 FB 143
BEGIN
   S704_LM_DC_PIN.Enable_Aux := FALSE;
   S704_LM_DC_PIN.Adv_Amount := 0;
   S704_LM_DC_PIN.Ret_Amount := 0;
   S704_LM_DC_PIN.LS_Adv1 := FALSE;
   S704_LM_DC_PIN.LS_Ret1 := FALSE;
   S704_LM_DC_PIN.LS_Adv2 := FALSE;
   S704_LM_DC_PIN.LS_Ret2 := FALSE;
   S704_LM_DC_PIN.LS_Adv3 := FALSE;
   S704_LM_DC_PIN.LS_Ret3 := FALSE;
   S704_LM_DC_PIN.LS_Adv4 := FALSE;
   S704_LM_DC_PIN.LS_Ret4 := FALSE;
   S704_LM_DC_PIN.SOL_Adv := FALSE;
   S704_LM_DC_PIN.SOL_Ret := FALSE;
   S704_LM_DC_PIN.M_Ready := FALSE;
   S704_LM_DC_PIN.T_CHK1 := T#0MS;
   S704_LM_DC_PIN.T_CHK2 := T#0MS;
   S704_LM_DC_PIN.PB_Lamp_CHK := FALSE;
   S704_LM_DC_PIN.PB_Error_Rst := FALSE;
   S704_LM_DC_PIN.M_FLICK := FALSE;
   S704_LM_DC_PIN.M_Adv_Err := FALSE;
   S704_LM_DC_PIN.M_Ret_Err := FALSE;
   S704_LM_DC_PIN.LP_Adv := FALSE;
   S704_LM_DC_PIN.LP_Ret := FALSE;
   S704_LM_DC_PIN.Visu_Adv := W#16#0;
   S704_LM_DC_PIN.Visu_Ret := W#16#0;
   S704_LM_DC_PIN.Error_T1.IN := FALSE;
   S704_LM_DC_PIN.Error_T1.PT := T#0MS;
   S704_LM_DC_PIN.Error_T1.Q := FALSE;
   S704_LM_DC_PIN.Error_T1.ET := T#0MS;
   S704_LM_DC_PIN.Error_T1.STATE := B#16#0;
   S704_LM_DC_PIN.Error_T1.STIME := T#0MS;
   S704_LM_DC_PIN.Error_T1.ATIME := T#0MS;
   S704_LM_DC_PIN.Error_T2.IN := FALSE;
   S704_LM_DC_PIN.Error_T2.PT := T#0MS;
   S704_LM_DC_PIN.Error_T2.Q := FALSE;
   S704_LM_DC_PIN.Error_T2.ET := T#0MS;
   S704_LM_DC_PIN.Error_T2.STATE := B#16#0;
   S704_LM_DC_PIN.Error_T2.STIME := T#0MS;
   S704_LM_DC_PIN.Error_T2.ATIME := T#0MS;
   S704_LM_DC_PIN.CHK_Aux1 := FALSE;
   S704_LM_DC_PIN.CHK_Aux2 := FALSE;
   S704_LM_DC_PIN.Error_T1_DN := FALSE;
   S704_LM_DC_PIN.Error_T2_DN := FALSE;
   S704_LM_DC_PIN.Adv_Memo := FALSE;
   S704_LM_DC_PIN.Visu_Adv_Arr[0] := FALSE;
   S704_LM_DC_PIN.Visu_Adv_Arr[1] := FALSE;
   S704_LM_DC_PIN.Visu_Adv_Arr[2] := FALSE;
   S704_LM_DC_PIN.Visu_Adv_Arr[3] := FALSE;
   S704_LM_DC_PIN.Visu_Adv_Arr[4] := FALSE;
   S704_LM_DC_PIN.Visu_Adv_Arr[5] := FALSE;
   S704_LM_DC_PIN.Visu_Adv_Arr[6] := FALSE;
   S704_LM_DC_PIN.Visu_Adv_Arr[7] := FALSE;
   S704_LM_DC_PIN.Visu_Adv_Arr[8] := FALSE;
   S704_LM_DC_PIN.Visu_Adv_Arr[9] := FALSE;
   S704_LM_DC_PIN.Visu_Adv_Arr[10] := FALSE;
   S704_LM_DC_PIN.Visu_Adv_Arr[11] := FALSE;
   S704_LM_DC_PIN.Visu_Adv_Arr[12] := FALSE;
   S704_LM_DC_PIN.Visu_Adv_Arr[13] := FALSE;
   S704_LM_DC_PIN.Visu_Adv_Arr[14] := FALSE;
   S704_LM_DC_PIN.Visu_Adv_Arr[15] := FALSE;
   S704_LM_DC_PIN.Visu_Ret_Arr[0] := FALSE;
   S704_LM_DC_PIN.Visu_Ret_Arr[1] := FALSE;
   S704_LM_DC_PIN.Visu_Ret_Arr[2] := FALSE;
   S704_LM_DC_PIN.Visu_Ret_Arr[3] := FALSE;
   S704_LM_DC_PIN.Visu_Ret_Arr[4] := FALSE;
   S704_LM_DC_PIN.Visu_Ret_Arr[5] := FALSE;
   S704_LM_DC_PIN.Visu_Ret_Arr[6] := FALSE;
   S704_LM_DC_PIN.Visu_Ret_Arr[7] := FALSE;
   S704_LM_DC_PIN.Visu_Ret_Arr[8] := FALSE;
   S704_LM_DC_PIN.Visu_Ret_Arr[9] := FALSE;
   S704_LM_DC_PIN.Visu_Ret_Arr[10] := FALSE;
   S704_LM_DC_PIN.Visu_Ret_Arr[11] := FALSE;
   S704_LM_DC_PIN.Visu_Ret_Arr[12] := FALSE;
   S704_LM_DC_PIN.Visu_Ret_Arr[13] := FALSE;
   S704_LM_DC_PIN.Visu_Ret_Arr[14] := FALSE;
   S704_LM_DC_PIN.Visu_Ret_Arr[15] := FALSE;
   S704_LM_DC_PIN.BLK_Move_Ret := 0;
   S704_LM_DC_PIN.Enable := FALSE;
   S704_LM_DC_PIN.Adv_End := FALSE;
   S704_LM_DC_PIN.Ret_End := FALSE;
   S704_LM_DC_1ST_CLAMP1.Enable_Aux := FALSE;
   S704_LM_DC_1ST_CLAMP1.Adv_Amount := 0;
   S704_LM_DC_1ST_CLAMP1.Ret_Amount := 0;
   S704_LM_DC_1ST_CLAMP1.LS_Adv1 := FALSE;
   S704_LM_DC_1ST_CLAMP1.LS_Ret1 := FALSE;
   S704_LM_DC_1ST_CLAMP1.LS_Adv2 := FALSE;
   S704_LM_DC_1ST_CLAMP1.LS_Ret2 := FALSE;
   S704_LM_DC_1ST_CLAMP1.LS_Adv3 := FALSE;
   S704_LM_DC_1ST_CLAMP1.LS_Ret3 := FALSE;
   S704_LM_DC_1ST_CLAMP1.LS_Adv4 := FALSE;
   S704_LM_DC_1ST_CLAMP1.LS_Ret4 := FALSE;
   S704_LM_DC_1ST_CLAMP1.SOL_Adv := FALSE;
   S704_LM_DC_1ST_CLAMP1.SOL_Ret := FALSE;
   S704_LM_DC_1ST_CLAMP1.M_Ready := FALSE;
   S704_LM_DC_1ST_CLAMP1.T_CHK1 := T#0MS;
   S704_LM_DC_1ST_CLAMP1.T_CHK2 := T#0MS;
   S704_LM_DC_1ST_CLAMP1.PB_Lamp_CHK := FALSE;
   S704_LM_DC_1ST_CLAMP1.PB_Error_Rst := FALSE;
   S704_LM_DC_1ST_CLAMP1.M_FLICK := FALSE;
   S704_LM_DC_1ST_CLAMP1.M_Adv_Err := FALSE;
   S704_LM_DC_1ST_CLAMP1.M_Ret_Err := FALSE;
   S704_LM_DC_1ST_CLAMP1.LP_Adv := FALSE;
   S704_LM_DC_1ST_CLAMP1.LP_Ret := FALSE;
   S704_LM_DC_1ST_CLAMP1.Visu_Adv := W#16#0;
   S704_LM_DC_1ST_CLAMP1.Visu_Ret := W#16#0;
   S704_LM_DC_1ST_CLAMP1.Error_T1.IN := FALSE;
   S704_LM_DC_1ST_CLAMP1.Error_T1.PT := T#0MS;
   S704_LM_DC_1ST_CLAMP1.Error_T1.Q := FALSE;
   S704_LM_DC_1ST_CLAMP1.Error_T1.ET := T#0MS;
   S704_LM_DC_1ST_CLAMP1.Error_T1.STATE := B#16#0;
   S704_LM_DC_1ST_CLAMP1.Error_T1.STIME := T#0MS;
   S704_LM_DC_1ST_CLAMP1.Error_T1.ATIME := T#0MS;
   S704_LM_DC_1ST_CLAMP1.Error_T2.IN := FALSE;
   S704_LM_DC_1ST_CLAMP1.Error_T2.PT := T#0MS;
   S704_LM_DC_1ST_CLAMP1.Error_T2.Q := FALSE;
   S704_LM_DC_1ST_CLAMP1.Error_T2.ET := T#0MS;
   S704_LM_DC_1ST_CLAMP1.Error_T2.STATE := B#16#0;
   S704_LM_DC_1ST_CLAMP1.Error_T2.STIME := T#0MS;
   S704_LM_DC_1ST_CLAMP1.Error_T2.ATIME := T#0MS;
   S704_LM_DC_1ST_CLAMP1.CHK_Aux1 := FALSE;
   S704_LM_DC_1ST_CLAMP1.CHK_Aux2 := FALSE;
   S704_LM_DC_1ST_CLAMP1.Error_T1_DN := FALSE;
   S704_LM_DC_1ST_CLAMP1.Error_T2_DN := FALSE;
   S704_LM_DC_1ST_CLAMP1.Adv_Memo := FALSE;
   S704_LM_DC_1ST_CLAMP1.Visu_Adv_Arr[0] := FALSE;
   S704_LM_DC_1ST_CLAMP1.Visu_Adv_Arr[1] := FALSE;
   S704_LM_DC_1ST_CLAMP1.Visu_Adv_Arr[2] := FALSE;
   S704_LM_DC_1ST_CLAMP1.Visu_Adv_Arr[3] := FALSE;
   S704_LM_DC_1ST_CLAMP1.Visu_Adv_Arr[4] := FALSE;
   S704_LM_DC_1ST_CLAMP1.Visu_Adv_Arr[5] := FALSE;
   S704_LM_DC_1ST_CLAMP1.Visu_Adv_Arr[6] := FALSE;
   S704_LM_DC_1ST_CLAMP1.Visu_Adv_Arr[7] := FALSE;
   S704_LM_DC_1ST_CLAMP1.Visu_Adv_Arr[8] := FALSE;
   S704_LM_DC_1ST_CLAMP1.Visu_Adv_Arr[9] := FALSE;
   S704_LM_DC_1ST_CLAMP1.Visu_Adv_Arr[10] := FALSE;
   S704_LM_DC_1ST_CLAMP1.Visu_Adv_Arr[11] := FALSE;
   S704_LM_DC_1ST_CLAMP1.Visu_Adv_Arr[12] := FALSE;
   S704_LM_DC_1ST_CLAMP1.Visu_Adv_Arr[13] := FALSE;
   S704_LM_DC_1ST_CLAMP1.Visu_Adv_Arr[14] := FALSE;
   S704_LM_DC_1ST_CLAMP1.Visu_Adv_Arr[15] := FALSE;
   S704_LM_DC_1ST_CLAMP1.Visu_Ret_Arr[0] := FALSE;
   S704_LM_DC_1ST_CLAMP1.Visu_Ret_Arr[1] := FALSE;
   S704_LM_DC_1ST_CLAMP1.Visu_Ret_Arr[2] := FALSE;
   S704_LM_DC_1ST_CLAMP1.Visu_Ret_Arr[3] := FALSE;
   S704_LM_DC_1ST_CLAMP1.Visu_Ret_Arr[4] := FALSE;
   S704_LM_DC_1ST_CLAMP1.Visu_Ret_Arr[5] := FALSE;
   S704_LM_DC_1ST_CLAMP1.Visu_Ret_Arr[6] := FALSE;
   S704_LM_DC_1ST_CLAMP1.Visu_Ret_Arr[7] := FALSE;
   S704_LM_DC_1ST_CLAMP1.Visu_Ret_Arr[8] := FALSE;
   S704_LM_DC_1ST_CLAMP1.Visu_Ret_Arr[9] := FALSE;
   S704_LM_DC_1ST_CLAMP1.Visu_Ret_Arr[10] := FALSE;
   S704_LM_DC_1ST_CLAMP1.Visu_Ret_Arr[11] := FALSE;
   S704_LM_DC_1ST_CLAMP1.Visu_Ret_Arr[12] := FALSE;
   S704_LM_DC_1ST_CLAMP1.Visu_Ret_Arr[13] := FALSE;
   S704_LM_DC_1ST_CLAMP1.Visu_Ret_Arr[14] := FALSE;
   S704_LM_DC_1ST_CLAMP1.Visu_Ret_Arr[15] := FALSE;
   S704_LM_DC_1ST_CLAMP1.BLK_Move_Ret := 0;
   S704_LM_DC_1ST_CLAMP1.Enable := FALSE;
   S704_LM_DC_1ST_CLAMP1.Adv_End := FALSE;
   S704_LM_DC_1ST_CLAMP1.Ret_End := FALSE;
   S704_LM_DC_1ST_CLAMP2.Enable_Aux := FALSE;
   S704_LM_DC_1ST_CLAMP2.Adv_Amount := 0;
   S704_LM_DC_1ST_CLAMP2.Ret_Amount := 0;
   S704_LM_DC_1ST_CLAMP2.LS_Adv1 := FALSE;
   S704_LM_DC_1ST_CLAMP2.LS_Ret1 := FALSE;
   S704_LM_DC_1ST_CLAMP2.LS_Adv2 := FALSE;
   S704_LM_DC_1ST_CLAMP2.LS_Ret2 := FALSE;
   S704_LM_DC_1ST_CLAMP2.LS_Adv3 := FALSE;
   S704_LM_DC_1ST_CLAMP2.LS_Ret3 := FALSE;
   S704_LM_DC_1ST_CLAMP2.LS_Adv4 := FALSE;
   S704_LM_DC_1ST_CLAMP2.LS_Ret4 := FALSE;
   S704_LM_DC_1ST_CLAMP2.SOL_Adv := FALSE;
   S704_LM_DC_1ST_CLAMP2.SOL_Ret := FALSE;
   S704_LM_DC_1ST_CLAMP2.M_Ready := FALSE;
   S704_LM_DC_1ST_CLAMP2.T_CHK1 := T#0MS;
   S704_LM_DC_1ST_CLAMP2.T_CHK2 := T#0MS;
   S704_LM_DC_1ST_CLAMP2.PB_Lamp_CHK := FALSE;
   S704_LM_DC_1ST_CLAMP2.PB_Error_Rst := FALSE;
   S704_LM_DC_1ST_CLAMP2.M_FLICK := FALSE;
   S704_LM_DC_1ST_CLAMP2.M_Adv_Err := FALSE;
   S704_LM_DC_1ST_CLAMP2.M_Ret_Err := FALSE;
   S704_LM_DC_1ST_CLAMP2.LP_Adv := FALSE;
   S704_LM_DC_1ST_CLAMP2.LP_Ret := FALSE;
   S704_LM_DC_1ST_CLAMP2.Visu_Adv := W#16#0;
   S704_LM_DC_1ST_CLAMP2.Visu_Ret := W#16#0;
   S704_LM_DC_1ST_CLAMP2.Error_T1.IN := FALSE;
   S704_LM_DC_1ST_CLAMP2.Error_T1.PT := T#0MS;
   S704_LM_DC_1ST_CLAMP2.Error_T1.Q := FALSE;
   S704_LM_DC_1ST_CLAMP2.Error_T1.ET := T#0MS;
   S704_LM_DC_1ST_CLAMP2.Error_T1.STATE := B#16#0;
   S704_LM_DC_1ST_CLAMP2.Error_T1.STIME := T#0MS;
   S704_LM_DC_1ST_CLAMP2.Error_T1.ATIME := T#0MS;
   S704_LM_DC_1ST_CLAMP2.Error_T2.IN := FALSE;
   S704_LM_DC_1ST_CLAMP2.Error_T2.PT := T#0MS;
   S704_LM_DC_1ST_CLAMP2.Error_T2.Q := FALSE;
   S704_LM_DC_1ST_CLAMP2.Error_T2.ET := T#0MS;
   S704_LM_DC_1ST_CLAMP2.Error_T2.STATE := B#16#0;
   S704_LM_DC_1ST_CLAMP2.Error_T2.STIME := T#0MS;
   S704_LM_DC_1ST_CLAMP2.Error_T2.ATIME := T#0MS;
   S704_LM_DC_1ST_CLAMP2.CHK_Aux1 := FALSE;
   S704_LM_DC_1ST_CLAMP2.CHK_Aux2 := FALSE;
   S704_LM_DC_1ST_CLAMP2.Error_T1_DN := FALSE;
   S704_LM_DC_1ST_CLAMP2.Error_T2_DN := FALSE;
   S704_LM_DC_1ST_CLAMP2.Adv_Memo := FALSE;
   S704_LM_DC_1ST_CLAMP2.Visu_Adv_Arr[0] := FALSE;
   S704_LM_DC_1ST_CLAMP2.Visu_Adv_Arr[1] := FALSE;
   S704_LM_DC_1ST_CLAMP2.Visu_Adv_Arr[2] := FALSE;
   S704_LM_DC_1ST_CLAMP2.Visu_Adv_Arr[3] := FALSE;
   S704_LM_DC_1ST_CLAMP2.Visu_Adv_Arr[4] := FALSE;
   S704_LM_DC_1ST_CLAMP2.Visu_Adv_Arr[5] := FALSE;
   S704_LM_DC_1ST_CLAMP2.Visu_Adv_Arr[6] := FALSE;
   S704_LM_DC_1ST_CLAMP2.Visu_Adv_Arr[7] := FALSE;
   S704_LM_DC_1ST_CLAMP2.Visu_Adv_Arr[8] := FALSE;
   S704_LM_DC_1ST_CLAMP2.Visu_Adv_Arr[9] := FALSE;
   S704_LM_DC_1ST_CLAMP2.Visu_Adv_Arr[10] := FALSE;
   S704_LM_DC_1ST_CLAMP2.Visu_Adv_Arr[11] := FALSE;
   S704_LM_DC_1ST_CLAMP2.Visu_Adv_Arr[12] := FALSE;
   S704_LM_DC_1ST_CLAMP2.Visu_Adv_Arr[13] := FALSE;
   S704_LM_DC_1ST_CLAMP2.Visu_Adv_Arr[14] := FALSE;
   S704_LM_DC_1ST_CLAMP2.Visu_Adv_Arr[15] := FALSE;
   S704_LM_DC_1ST_CLAMP2.Visu_Ret_Arr[0] := FALSE;
   S704_LM_DC_1ST_CLAMP2.Visu_Ret_Arr[1] := FALSE;
   S704_LM_DC_1ST_CLAMP2.Visu_Ret_Arr[2] := FALSE;
   S704_LM_DC_1ST_CLAMP2.Visu_Ret_Arr[3] := FALSE;
   S704_LM_DC_1ST_CLAMP2.Visu_Ret_Arr[4] := FALSE;
   S704_LM_DC_1ST_CLAMP2.Visu_Ret_Arr[5] := FALSE;
   S704_LM_DC_1ST_CLAMP2.Visu_Ret_Arr[6] := FALSE;
   S704_LM_DC_1ST_CLAMP2.Visu_Ret_Arr[7] := FALSE;
   S704_LM_DC_1ST_CLAMP2.Visu_Ret_Arr[8] := FALSE;
   S704_LM_DC_1ST_CLAMP2.Visu_Ret_Arr[9] := FALSE;
   S704_LM_DC_1ST_CLAMP2.Visu_Ret_Arr[10] := FALSE;
   S704_LM_DC_1ST_CLAMP2.Visu_Ret_Arr[11] := FALSE;
   S704_LM_DC_1ST_CLAMP2.Visu_Ret_Arr[12] := FALSE;
   S704_LM_DC_1ST_CLAMP2.Visu_Ret_Arr[13] := FALSE;
   S704_LM_DC_1ST_CLAMP2.Visu_Ret_Arr[14] := FALSE;
   S704_LM_DC_1ST_CLAMP2.Visu_Ret_Arr[15] := FALSE;
   S704_LM_DC_1ST_CLAMP2.BLK_Move_Ret := 0;
   S704_LM_DC_1ST_CLAMP2.Enable := FALSE;
   S704_LM_DC_1ST_CLAMP2.Adv_End := FALSE;
   S704_LM_DC_1ST_CLAMP2.Ret_End := FALSE;
   S704_LM_DC_1ST_CLAMP3.Enable_Aux := FALSE;
   S704_LM_DC_1ST_CLAMP3.Adv_Amount := 0;
   S704_LM_DC_1ST_CLAMP3.Ret_Amount := 0;
   S704_LM_DC_1ST_CLAMP3.LS_Adv1 := FALSE;
   S704_LM_DC_1ST_CLAMP3.LS_Ret1 := FALSE;
   S704_LM_DC_1ST_CLAMP3.LS_Adv2 := FALSE;
   S704_LM_DC_1ST_CLAMP3.LS_Ret2 := FALSE;
   S704_LM_DC_1ST_CLAMP3.LS_Adv3 := FALSE;
   S704_LM_DC_1ST_CLAMP3.LS_Ret3 := FALSE;
   S704_LM_DC_1ST_CLAMP3.LS_Adv4 := FALSE;
   S704_LM_DC_1ST_CLAMP3.LS_Ret4 := FALSE;
   S704_LM_DC_1ST_CLAMP3.SOL_Adv := FALSE;
   S704_LM_DC_1ST_CLAMP3.SOL_Ret := FALSE;
   S704_LM_DC_1ST_CLAMP3.M_Ready := FALSE;
   S704_LM_DC_1ST_CLAMP3.T_CHK1 := T#0MS;
   S704_LM_DC_1ST_CLAMP3.T_CHK2 := T#0MS;
   S704_LM_DC_1ST_CLAMP3.PB_Lamp_CHK := FALSE;
   S704_LM_DC_1ST_CLAMP3.PB_Error_Rst := FALSE;
   S704_LM_DC_1ST_CLAMP3.M_FLICK := FALSE;
   S704_LM_DC_1ST_CLAMP3.M_Adv_Err := FALSE;
   S704_LM_DC_1ST_CLAMP3.M_Ret_Err := FALSE;
   S704_LM_DC_1ST_CLAMP3.LP_Adv := FALSE;
   S704_LM_DC_1ST_CLAMP3.LP_Ret := FALSE;
   S704_LM_DC_1ST_CLAMP3.Visu_Adv := W#16#0;
   S704_LM_DC_1ST_CLAMP3.Visu_Ret := W#16#0;
   S704_LM_DC_1ST_CLAMP3.Error_T1.IN := FALSE;
   S704_LM_DC_1ST_CLAMP3.Error_T1.PT := T#0MS;
   S704_LM_DC_1ST_CLAMP3.Error_T1.Q := FALSE;
   S704_LM_DC_1ST_CLAMP3.Error_T1.ET := T#0MS;
   S704_LM_DC_1ST_CLAMP3.Error_T1.STATE := B#16#0;
   S704_LM_DC_1ST_CLAMP3.Error_T1.STIME := T#0MS;
   S704_LM_DC_1ST_CLAMP3.Error_T1.ATIME := T#0MS;
   S704_LM_DC_1ST_CLAMP3.Error_T2.IN := FALSE;
   S704_LM_DC_1ST_CLAMP3.Error_T2.PT := T#0MS;
   S704_LM_DC_1ST_CLAMP3.Error_T2.Q := FALSE;
   S704_LM_DC_1ST_CLAMP3.Error_T2.ET := T#0MS;
   S704_LM_DC_1ST_CLAMP3.Error_T2.STATE := B#16#0;
   S704_LM_DC_1ST_CLAMP3.Error_T2.STIME := T#0MS;
   S704_LM_DC_1ST_CLAMP3.Error_T2.ATIME := T#0MS;
   S704_LM_DC_1ST_CLAMP3.CHK_Aux1 := FALSE;
   S704_LM_DC_1ST_CLAMP3.CHK_Aux2 := FALSE;
   S704_LM_DC_1ST_CLAMP3.Error_T1_DN := FALSE;
   S704_LM_DC_1ST_CLAMP3.Error_T2_DN := FALSE;
   S704_LM_DC_1ST_CLAMP3.Adv_Memo := FALSE;
   S704_LM_DC_1ST_CLAMP3.Visu_Adv_Arr[0] := FALSE;
   S704_LM_DC_1ST_CLAMP3.Visu_Adv_Arr[1] := FALSE;
   S704_LM_DC_1ST_CLAMP3.Visu_Adv_Arr[2] := FALSE;
   S704_LM_DC_1ST_CLAMP3.Visu_Adv_Arr[3] := FALSE;
   S704_LM_DC_1ST_CLAMP3.Visu_Adv_Arr[4] := FALSE;
   S704_LM_DC_1ST_CLAMP3.Visu_Adv_Arr[5] := FALSE;
   S704_LM_DC_1ST_CLAMP3.Visu_Adv_Arr[6] := FALSE;
   S704_LM_DC_1ST_CLAMP3.Visu_Adv_Arr[7] := FALSE;
   S704_LM_DC_1ST_CLAMP3.Visu_Adv_Arr[8] := FALSE;
   S704_LM_DC_1ST_CLAMP3.Visu_Adv_Arr[9] := FALSE;
   S704_LM_DC_1ST_CLAMP3.Visu_Adv_Arr[10] := FALSE;
   S704_LM_DC_1ST_CLAMP3.Visu_Adv_Arr[11] := FALSE;
   S704_LM_DC_1ST_CLAMP3.Visu_Adv_Arr[12] := FALSE;
   S704_LM_DC_1ST_CLAMP3.Visu_Adv_Arr[13] := FALSE;
   S704_LM_DC_1ST_CLAMP3.Visu_Adv_Arr[14] := FALSE;
   S704_LM_DC_1ST_CLAMP3.Visu_Adv_Arr[15] := FALSE;
   S704_LM_DC_1ST_CLAMP3.Visu_Ret_Arr[0] := FALSE;
   S704_LM_DC_1ST_CLAMP3.Visu_Ret_Arr[1] := FALSE;
   S704_LM_DC_1ST_CLAMP3.Visu_Ret_Arr[2] := FALSE;
   S704_LM_DC_1ST_CLAMP3.Visu_Ret_Arr[3] := FALSE;
   S704_LM_DC_1ST_CLAMP3.Visu_Ret_Arr[4] := FALSE;
   S704_LM_DC_1ST_CLAMP3.Visu_Ret_Arr[5] := FALSE;
   S704_LM_DC_1ST_CLAMP3.Visu_Ret_Arr[6] := FALSE;
   S704_LM_DC_1ST_CLAMP3.Visu_Ret_Arr[7] := FALSE;
   S704_LM_DC_1ST_CLAMP3.Visu_Ret_Arr[8] := FALSE;
   S704_LM_DC_1ST_CLAMP3.Visu_Ret_Arr[9] := FALSE;
   S704_LM_DC_1ST_CLAMP3.Visu_Ret_Arr[10] := FALSE;
   S704_LM_DC_1ST_CLAMP3.Visu_Ret_Arr[11] := FALSE;
   S704_LM_DC_1ST_CLAMP3.Visu_Ret_Arr[12] := FALSE;
   S704_LM_DC_1ST_CLAMP3.Visu_Ret_Arr[13] := FALSE;
   S704_LM_DC_1ST_CLAMP3.Visu_Ret_Arr[14] := FALSE;
   S704_LM_DC_1ST_CLAMP3.Visu_Ret_Arr[15] := FALSE;
   S704_LM_DC_1ST_CLAMP3.BLK_Move_Ret := 0;
   S704_LM_DC_1ST_CLAMP3.Enable := FALSE;
   S704_LM_DC_1ST_CLAMP3.Adv_End := FALSE;
   S704_LM_DC_1ST_CLAMP3.Ret_End := FALSE;
   S704_LM_DC_1ST_CLAMP4.Enable_Aux := FALSE;
   S704_LM_DC_1ST_CLAMP4.Adv_Amount := 0;
   S704_LM_DC_1ST_CLAMP4.Ret_Amount := 0;
   S704_LM_DC_1ST_CLAMP4.LS_Adv1 := FALSE;
   S704_LM_DC_1ST_CLAMP4.LS_Ret1 := FALSE;
   S704_LM_DC_1ST_CLAMP4.LS_Adv2 := FALSE;
   S704_LM_DC_1ST_CLAMP4.LS_Ret2 := FALSE;
   S704_LM_DC_1ST_CLAMP4.LS_Adv3 := FALSE;
   S704_LM_DC_1ST_CLAMP4.LS_Ret3 := FALSE;
   S704_LM_DC_1ST_CLAMP4.LS_Adv4 := FALSE;
   S704_LM_DC_1ST_CLAMP4.LS_Ret4 := FALSE;
   S704_LM_DC_1ST_CLAMP4.SOL_Adv := FALSE;
   S704_LM_DC_1ST_CLAMP4.SOL_Ret := FALSE;
   S704_LM_DC_1ST_CLAMP4.M_Ready := FALSE;
   S704_LM_DC_1ST_CLAMP4.T_CHK1 := T#0MS;
   S704_LM_DC_1ST_CLAMP4.T_CHK2 := T#0MS;
   S704_LM_DC_1ST_CLAMP4.PB_Lamp_CHK := FALSE;
   S704_LM_DC_1ST_CLAMP4.PB_Error_Rst := FALSE;
   S704_LM_DC_1ST_CLAMP4.M_FLICK := FALSE;
   S704_LM_DC_1ST_CLAMP4.M_Adv_Err := FALSE;
   S704_LM_DC_1ST_CLAMP4.M_Ret_Err := FALSE;
   S704_LM_DC_1ST_CLAMP4.LP_Adv := FALSE;
   S704_LM_DC_1ST_CLAMP4.LP_Ret := FALSE;
   S704_LM_DC_1ST_CLAMP4.Visu_Adv := W#16#0;
   S704_LM_DC_1ST_CLAMP4.Visu_Ret := W#16#0;
   S704_LM_DC_1ST_CLAMP4.Error_T1.IN := FALSE;
   S704_LM_DC_1ST_CLAMP4.Error_T1.PT := T#0MS;
   S704_LM_DC_1ST_CLAMP4.Error_T1.Q := FALSE;
   S704_LM_DC_1ST_CLAMP4.Error_T1.ET := T#0MS;
   S704_LM_DC_1ST_CLAMP4.Error_T1.STATE := B#16#0;
   S704_LM_DC_1ST_CLAMP4.Error_T1.STIME := T#0MS;
   S704_LM_DC_1ST_CLAMP4.Error_T1.ATIME := T#0MS;
   S704_LM_DC_1ST_CLAMP4.Error_T2.IN := FALSE;
   S704_LM_DC_1ST_CLAMP4.Error_T2.PT := T#0MS;
   S704_LM_DC_1ST_CLAMP4.Error_T2.Q := FALSE;
   S704_LM_DC_1ST_CLAMP4.Error_T2.ET := T#0MS;
   S704_LM_DC_1ST_CLAMP4.Error_T2.STATE := B#16#0;
   S704_LM_DC_1ST_CLAMP4.Error_T2.STIME := T#0MS;
   S704_LM_DC_1ST_CLAMP4.Error_T2.ATIME := T#0MS;
   S704_LM_DC_1ST_CLAMP4.CHK_Aux1 := FALSE;
   S704_LM_DC_1ST_CLAMP4.CHK_Aux2 := FALSE;
   S704_LM_DC_1ST_CLAMP4.Error_T1_DN := FALSE;
   S704_LM_DC_1ST_CLAMP4.Error_T2_DN := FALSE;
   S704_LM_DC_1ST_CLAMP4.Adv_Memo := FALSE;
   S704_LM_DC_1ST_CLAMP4.Visu_Adv_Arr[0] := FALSE;
   S704_LM_DC_1ST_CLAMP4.Visu_Adv_Arr[1] := FALSE;
   S704_LM_DC_1ST_CLAMP4.Visu_Adv_Arr[2] := FALSE;
   S704_LM_DC_1ST_CLAMP4.Visu_Adv_Arr[3] := FALSE;
   S704_LM_DC_1ST_CLAMP4.Visu_Adv_Arr[4] := FALSE;
   S704_LM_DC_1ST_CLAMP4.Visu_Adv_Arr[5] := FALSE;
   S704_LM_DC_1ST_CLAMP4.Visu_Adv_Arr[6] := FALSE;
   S704_LM_DC_1ST_CLAMP4.Visu_Adv_Arr[7] := FALSE;
   S704_LM_DC_1ST_CLAMP4.Visu_Adv_Arr[8] := FALSE;
   S704_LM_DC_1ST_CLAMP4.Visu_Adv_Arr[9] := FALSE;
   S704_LM_DC_1ST_CLAMP4.Visu_Adv_Arr[10] := FALSE;
   S704_LM_DC_1ST_CLAMP4.Visu_Adv_Arr[11] := FALSE;
   S704_LM_DC_1ST_CLAMP4.Visu_Adv_Arr[12] := FALSE;
   S704_LM_DC_1ST_CLAMP4.Visu_Adv_Arr[13] := FALSE;
   S704_LM_DC_1ST_CLAMP4.Visu_Adv_Arr[14] := FALSE;
   S704_LM_DC_1ST_CLAMP4.Visu_Adv_Arr[15] := FALSE;
   S704_LM_DC_1ST_CLAMP4.Visu_Ret_Arr[0] := FALSE;
   S704_LM_DC_1ST_CLAMP4.Visu_Ret_Arr[1] := FALSE;
   S704_LM_DC_1ST_CLAMP4.Visu_Ret_Arr[2] := FALSE;
   S704_LM_DC_1ST_CLAMP4.Visu_Ret_Arr[3] := FALSE;
   S704_LM_DC_1ST_CLAMP4.Visu_Ret_Arr[4] := FALSE;
   S704_LM_DC_1ST_CLAMP4.Visu_Ret_Arr[5] := FALSE;
   S704_LM_DC_1ST_CLAMP4.Visu_Ret_Arr[6] := FALSE;
   S704_LM_DC_1ST_CLAMP4.Visu_Ret_Arr[7] := FALSE;
   S704_LM_DC_1ST_CLAMP4.Visu_Ret_Arr[8] := FALSE;
   S704_LM_DC_1ST_CLAMP4.Visu_Ret_Arr[9] := FALSE;
   S704_LM_DC_1ST_CLAMP4.Visu_Ret_Arr[10] := FALSE;
   S704_LM_DC_1ST_CLAMP4.Visu_Ret_Arr[11] := FALSE;
   S704_LM_DC_1ST_CLAMP4.Visu_Ret_Arr[12] := FALSE;
   S704_LM_DC_1ST_CLAMP4.Visu_Ret_Arr[13] := FALSE;
   S704_LM_DC_1ST_CLAMP4.Visu_Ret_Arr[14] := FALSE;
   S704_LM_DC_1ST_CLAMP4.Visu_Ret_Arr[15] := FALSE;
   S704_LM_DC_1ST_CLAMP4.BLK_Move_Ret := 0;
   S704_LM_DC_1ST_CLAMP4.Enable := FALSE;
   S704_LM_DC_1ST_CLAMP4.Adv_End := FALSE;
   S704_LM_DC_1ST_CLAMP4.Ret_End := FALSE;
   S704_LM_DC_2ND_CLAMP1.Enable_Aux := FALSE;
   S704_LM_DC_2ND_CLAMP1.Adv_Amount := 0;
   S704_LM_DC_2ND_CLAMP1.Ret_Amount := 0;
   S704_LM_DC_2ND_CLAMP1.LS_Adv1 := FALSE;
   S704_LM_DC_2ND_CLAMP1.LS_Ret1 := FALSE;
   S704_LM_DC_2ND_CLAMP1.LS_Adv2 := FALSE;
   S704_LM_DC_2ND_CLAMP1.LS_Ret2 := FALSE;
   S704_LM_DC_2ND_CLAMP1.LS_Adv3 := FALSE;
   S704_LM_DC_2ND_CLAMP1.LS_Ret3 := FALSE;
   S704_LM_DC_2ND_CLAMP1.LS_Adv4 := FALSE;
   S704_LM_DC_2ND_CLAMP1.LS_Ret4 := FALSE;
   S704_LM_DC_2ND_CLAMP1.SOL_Adv := FALSE;
   S704_LM_DC_2ND_CLAMP1.SOL_Ret := FALSE;
   S704_LM_DC_2ND_CLAMP1.M_Ready := FALSE;
   S704_LM_DC_2ND_CLAMP1.T_CHK1 := T#0MS;
   S704_LM_DC_2ND_CLAMP1.T_CHK2 := T#0MS;
   S704_LM_DC_2ND_CLAMP1.PB_Lamp_CHK := FALSE;
   S704_LM_DC_2ND_CLAMP1.PB_Error_Rst := FALSE;
   S704_LM_DC_2ND_CLAMP1.M_FLICK := FALSE;
   S704_LM_DC_2ND_CLAMP1.M_Adv_Err := FALSE;
   S704_LM_DC_2ND_CLAMP1.M_Ret_Err := FALSE;
   S704_LM_DC_2ND_CLAMP1.LP_Adv := FALSE;
   S704_LM_DC_2ND_CLAMP1.LP_Ret := FALSE;
   S704_LM_DC_2ND_CLAMP1.Visu_Adv := W#16#0;
   S704_LM_DC_2ND_CLAMP1.Visu_Ret := W#16#0;
   S704_LM_DC_2ND_CLAMP1.Error_T1.IN := FALSE;
   S704_LM_DC_2ND_CLAMP1.Error_T1.PT := T#0MS;
   S704_LM_DC_2ND_CLAMP1.Error_T1.Q := FALSE;
   S704_LM_DC_2ND_CLAMP1.Error_T1.ET := T#0MS;
   S704_LM_DC_2ND_CLAMP1.Error_T1.STATE := B#16#0;
   S704_LM_DC_2ND_CLAMP1.Error_T1.STIME := T#0MS;
   S704_LM_DC_2ND_CLAMP1.Error_T1.ATIME := T#0MS;
   S704_LM_DC_2ND_CLAMP1.Error_T2.IN := FALSE;
   S704_LM_DC_2ND_CLAMP1.Error_T2.PT := T#0MS;
   S704_LM_DC_2ND_CLAMP1.Error_T2.Q := FALSE;
   S704_LM_DC_2ND_CLAMP1.Error_T2.ET := T#0MS;
   S704_LM_DC_2ND_CLAMP1.Error_T2.STATE := B#16#0;
   S704_LM_DC_2ND_CLAMP1.Error_T2.STIME := T#0MS;
   S704_LM_DC_2ND_CLAMP1.Error_T2.ATIME := T#0MS;
   S704_LM_DC_2ND_CLAMP1.CHK_Aux1 := FALSE;
   S704_LM_DC_2ND_CLAMP1.CHK_Aux2 := FALSE;
   S704_LM_DC_2ND_CLAMP1.Error_T1_DN := FALSE;
   S704_LM_DC_2ND_CLAMP1.Error_T2_DN := FALSE;
   S704_LM_DC_2ND_CLAMP1.Adv_Memo := FALSE;
   S704_LM_DC_2ND_CLAMP1.Visu_Adv_Arr[0] := FALSE;
   S704_LM_DC_2ND_CLAMP1.Visu_Adv_Arr[1] := FALSE;
   S704_LM_DC_2ND_CLAMP1.Visu_Adv_Arr[2] := FALSE;
   S704_LM_DC_2ND_CLAMP1.Visu_Adv_Arr[3] := FALSE;
   S704_LM_DC_2ND_CLAMP1.Visu_Adv_Arr[4] := FALSE;
   S704_LM_DC_2ND_CLAMP1.Visu_Adv_Arr[5] := FALSE;
   S704_LM_DC_2ND_CLAMP1.Visu_Adv_Arr[6] := FALSE;
   S704_LM_DC_2ND_CLAMP1.Visu_Adv_Arr[7] := FALSE;
   S704_LM_DC_2ND_CLAMP1.Visu_Adv_Arr[8] := FALSE;
   S704_LM_DC_2ND_CLAMP1.Visu_Adv_Arr[9] := FALSE;
   S704_LM_DC_2ND_CLAMP1.Visu_Adv_Arr[10] := FALSE;
   S704_LM_DC_2ND_CLAMP1.Visu_Adv_Arr[11] := FALSE;
   S704_LM_DC_2ND_CLAMP1.Visu_Adv_Arr[12] := FALSE;
   S704_LM_DC_2ND_CLAMP1.Visu_Adv_Arr[13] := FALSE;
   S704_LM_DC_2ND_CLAMP1.Visu_Adv_Arr[14] := FALSE;
   S704_LM_DC_2ND_CLAMP1.Visu_Adv_Arr[15] := FALSE;
   S704_LM_DC_2ND_CLAMP1.Visu_Ret_Arr[0] := FALSE;
   S704_LM_DC_2ND_CLAMP1.Visu_Ret_Arr[1] := FALSE;
   S704_LM_DC_2ND_CLAMP1.Visu_Ret_Arr[2] := FALSE;
   S704_LM_DC_2ND_CLAMP1.Visu_Ret_Arr[3] := FALSE;
   S704_LM_DC_2ND_CLAMP1.Visu_Ret_Arr[4] := FALSE;
   S704_LM_DC_2ND_CLAMP1.Visu_Ret_Arr[5] := FALSE;
   S704_LM_DC_2ND_CLAMP1.Visu_Ret_Arr[6] := FALSE;
   S704_LM_DC_2ND_CLAMP1.Visu_Ret_Arr[7] := FALSE;
   S704_LM_DC_2ND_CLAMP1.Visu_Ret_Arr[8] := FALSE;
   S704_LM_DC_2ND_CLAMP1.Visu_Ret_Arr[9] := FALSE;
   S704_LM_DC_2ND_CLAMP1.Visu_Ret_Arr[10] := FALSE;
   S704_LM_DC_2ND_CLAMP1.Visu_Ret_Arr[11] := FALSE;
   S704_LM_DC_2ND_CLAMP1.Visu_Ret_Arr[12] := FALSE;
   S704_LM_DC_2ND_CLAMP1.Visu_Ret_Arr[13] := FALSE;
   S704_LM_DC_2ND_CLAMP1.Visu_Ret_Arr[14] := FALSE;
   S704_LM_DC_2ND_CLAMP1.Visu_Ret_Arr[15] := FALSE;
   S704_LM_DC_2ND_CLAMP1.BLK_Move_Ret := 0;
   S704_LM_DC_2ND_CLAMP1.Enable := FALSE;
   S704_LM_DC_2ND_CLAMP1.Adv_End := FALSE;
   S704_LM_DC_2ND_CLAMP1.Ret_End := FALSE;
   S704_LM_DC_2ND_CLAMP2.Enable_Aux := FALSE;
   S704_LM_DC_2ND_CLAMP2.Adv_Amount := 0;
   S704_LM_DC_2ND_CLAMP2.Ret_Amount := 0;
   S704_LM_DC_2ND_CLAMP2.LS_Adv1 := FALSE;
   S704_LM_DC_2ND_CLAMP2.LS_Ret1 := FALSE;
   S704_LM_DC_2ND_CLAMP2.LS_Adv2 := FALSE;
   S704_LM_DC_2ND_CLAMP2.LS_Ret2 := FALSE;
   S704_LM_DC_2ND_CLAMP2.LS_Adv3 := FALSE;
   S704_LM_DC_2ND_CLAMP2.LS_Ret3 := FALSE;
   S704_LM_DC_2ND_CLAMP2.LS_Adv4 := FALSE;
   S704_LM_DC_2ND_CLAMP2.LS_Ret4 := FALSE;
   S704_LM_DC_2ND_CLAMP2.SOL_Adv := FALSE;
   S704_LM_DC_2ND_CLAMP2.SOL_Ret := FALSE;
   S704_LM_DC_2ND_CLAMP2.M_Ready := FALSE;
   S704_LM_DC_2ND_CLAMP2.T_CHK1 := T#0MS;
   S704_LM_DC_2ND_CLAMP2.T_CHK2 := T#0MS;
   S704_LM_DC_2ND_CLAMP2.PB_Lamp_CHK := FALSE;
   S704_LM_DC_2ND_CLAMP2.PB_Error_Rst := FALSE;
   S704_LM_DC_2ND_CLAMP2.M_FLICK := FALSE;
   S704_LM_DC_2ND_CLAMP2.M_Adv_Err := FALSE;
   S704_LM_DC_2ND_CLAMP2.M_Ret_Err := FALSE;
   S704_LM_DC_2ND_CLAMP2.LP_Adv := FALSE;
   S704_LM_DC_2ND_CLAMP2.LP_Ret := FALSE;
   S704_LM_DC_2ND_CLAMP2.Visu_Adv := W#16#0;
   S704_LM_DC_2ND_CLAMP2.Visu_Ret := W#16#0;
   S704_LM_DC_2ND_CLAMP2.Error_T1.IN := FALSE;
   S704_LM_DC_2ND_CLAMP2.Error_T1.PT := T#0MS;
   S704_LM_DC_2ND_CLAMP2.Error_T1.Q := FALSE;
   S704_LM_DC_2ND_CLAMP2.Error_T1.ET := T#0MS;
   S704_LM_DC_2ND_CLAMP2.Error_T1.STATE := B#16#0;
   S704_LM_DC_2ND_CLAMP2.Error_T1.STIME := T#0MS;
   S704_LM_DC_2ND_CLAMP2.Error_T1.ATIME := T#0MS;
   S704_LM_DC_2ND_CLAMP2.Error_T2.IN := FALSE;
   S704_LM_DC_2ND_CLAMP2.Error_T2.PT := T#0MS;
   S704_LM_DC_2ND_CLAMP2.Error_T2.Q := FALSE;
   S704_LM_DC_2ND_CLAMP2.Error_T2.ET := T#0MS;
   S704_LM_DC_2ND_CLAMP2.Error_T2.STATE := B#16#0;
   S704_LM_DC_2ND_CLAMP2.Error_T2.STIME := T#0MS;
   S704_LM_DC_2ND_CLAMP2.Error_T2.ATIME := T#0MS;
   S704_LM_DC_2ND_CLAMP2.CHK_Aux1 := FALSE;
   S704_LM_DC_2ND_CLAMP2.CHK_Aux2 := FALSE;
   S704_LM_DC_2ND_CLAMP2.Error_T1_DN := FALSE;
   S704_LM_DC_2ND_CLAMP2.Error_T2_DN := FALSE;
   S704_LM_DC_2ND_CLAMP2.Adv_Memo := FALSE;
   S704_LM_DC_2ND_CLAMP2.Visu_Adv_Arr[0] := FALSE;
   S704_LM_DC_2ND_CLAMP2.Visu_Adv_Arr[1] := FALSE;
   S704_LM_DC_2ND_CLAMP2.Visu_Adv_Arr[2] := FALSE;
   S704_LM_DC_2ND_CLAMP2.Visu_Adv_Arr[3] := FALSE;
   S704_LM_DC_2ND_CLAMP2.Visu_Adv_Arr[4] := FALSE;
   S704_LM_DC_2ND_CLAMP2.Visu_Adv_Arr[5] := FALSE;
   S704_LM_DC_2ND_CLAMP2.Visu_Adv_Arr[6] := FALSE;
   S704_LM_DC_2ND_CLAMP2.Visu_Adv_Arr[7] := FALSE;
   S704_LM_DC_2ND_CLAMP2.Visu_Adv_Arr[8] := FALSE;
   S704_LM_DC_2ND_CLAMP2.Visu_Adv_Arr[9] := FALSE;
   S704_LM_DC_2ND_CLAMP2.Visu_Adv_Arr[10] := FALSE;
   S704_LM_DC_2ND_CLAMP2.Visu_Adv_Arr[11] := FALSE;
   S704_LM_DC_2ND_CLAMP2.Visu_Adv_Arr[12] := FALSE;
   S704_LM_DC_2ND_CLAMP2.Visu_Adv_Arr[13] := FALSE;
   S704_LM_DC_2ND_CLAMP2.Visu_Adv_Arr[14] := FALSE;
   S704_LM_DC_2ND_CLAMP2.Visu_Adv_Arr[15] := FALSE;
   S704_LM_DC_2ND_CLAMP2.Visu_Ret_Arr[0] := FALSE;
   S704_LM_DC_2ND_CLAMP2.Visu_Ret_Arr[1] := FALSE;
   S704_LM_DC_2ND_CLAMP2.Visu_Ret_Arr[2] := FALSE;
   S704_LM_DC_2ND_CLAMP2.Visu_Ret_Arr[3] := FALSE;
   S704_LM_DC_2ND_CLAMP2.Visu_Ret_Arr[4] := FALSE;
   S704_LM_DC_2ND_CLAMP2.Visu_Ret_Arr[5] := FALSE;
   S704_LM_DC_2ND_CLAMP2.Visu_Ret_Arr[6] := FALSE;
   S704_LM_DC_2ND_CLAMP2.Visu_Ret_Arr[7] := FALSE;
   S704_LM_DC_2ND_CLAMP2.Visu_Ret_Arr[8] := FALSE;
   S704_LM_DC_2ND_CLAMP2.Visu_Ret_Arr[9] := FALSE;
   S704_LM_DC_2ND_CLAMP2.Visu_Ret_Arr[10] := FALSE;
   S704_LM_DC_2ND_CLAMP2.Visu_Ret_Arr[11] := FALSE;
   S704_LM_DC_2ND_CLAMP2.Visu_Ret_Arr[12] := FALSE;
   S704_LM_DC_2ND_CLAMP2.Visu_Ret_Arr[13] := FALSE;
   S704_LM_DC_2ND_CLAMP2.Visu_Ret_Arr[14] := FALSE;
   S704_LM_DC_2ND_CLAMP2.Visu_Ret_Arr[15] := FALSE;
   S704_LM_DC_2ND_CLAMP2.BLK_Move_Ret := 0;
   S704_LM_DC_2ND_CLAMP2.Enable := FALSE;
   S704_LM_DC_2ND_CLAMP2.Adv_End := FALSE;
   S704_LM_DC_2ND_CLAMP2.Ret_End := FALSE;
   S704_LM_DC_2ND_CLAMP3.Enable_Aux := FALSE;
   S704_LM_DC_2ND_CLAMP3.Adv_Amount := 0;
   S704_LM_DC_2ND_CLAMP3.Ret_Amount := 0;
   S704_LM_DC_2ND_CLAMP3.LS_Adv1 := FALSE;
   S704_LM_DC_2ND_CLAMP3.LS_Ret1 := FALSE;
   S704_LM_DC_2ND_CLAMP3.LS_Adv2 := FALSE;
   S704_LM_DC_2ND_CLAMP3.LS_Ret2 := FALSE;
   S704_LM_DC_2ND_CLAMP3.LS_Adv3 := FALSE;
   S704_LM_DC_2ND_CLAMP3.LS_Ret3 := FALSE;
   S704_LM_DC_2ND_CLAMP3.LS_Adv4 := FALSE;
   S704_LM_DC_2ND_CLAMP3.LS_Ret4 := FALSE;
   S704_LM_DC_2ND_CLAMP3.SOL_Adv := FALSE;
   S704_LM_DC_2ND_CLAMP3.SOL_Ret := FALSE;
   S704_LM_DC_2ND_CLAMP3.M_Ready := FALSE;
   S704_LM_DC_2ND_CLAMP3.T_CHK1 := T#0MS;
   S704_LM_DC_2ND_CLAMP3.T_CHK2 := T#0MS;
   S704_LM_DC_2ND_CLAMP3.PB_Lamp_CHK := FALSE;
   S704_LM_DC_2ND_CLAMP3.PB_Error_Rst := FALSE;
   S704_LM_DC_2ND_CLAMP3.M_FLICK := FALSE;
   S704_LM_DC_2ND_CLAMP3.M_Adv_Err := FALSE;
   S704_LM_DC_2ND_CLAMP3.M_Ret_Err := FALSE;
   S704_LM_DC_2ND_CLAMP3.LP_Adv := FALSE;
   S704_LM_DC_2ND_CLAMP3.LP_Ret := FALSE;
   S704_LM_DC_2ND_CLAMP3.Visu_Adv := W#16#0;
   S704_LM_DC_2ND_CLAMP3.Visu_Ret := W#16#0;
   S704_LM_DC_2ND_CLAMP3.Error_T1.IN := FALSE;
   S704_LM_DC_2ND_CLAMP3.Error_T1.PT := T#0MS;
   S704_LM_DC_2ND_CLAMP3.Error_T1.Q := FALSE;
   S704_LM_DC_2ND_CLAMP3.Error_T1.ET := T#0MS;
   S704_LM_DC_2ND_CLAMP3.Error_T1.STATE := B#16#0;
   S704_LM_DC_2ND_CLAMP3.Error_T1.STIME := T#0MS;
   S704_LM_DC_2ND_CLAMP3.Error_T1.ATIME := T#0MS;
   S704_LM_DC_2ND_CLAMP3.Error_T2.IN := FALSE;
   S704_LM_DC_2ND_CLAMP3.Error_T2.PT := T#0MS;
   S704_LM_DC_2ND_CLAMP3.Error_T2.Q := FALSE;
   S704_LM_DC_2ND_CLAMP3.Error_T2.ET := T#0MS;
   S704_LM_DC_2ND_CLAMP3.Error_T2.STATE := B#16#0;
   S704_LM_DC_2ND_CLAMP3.Error_T2.STIME := T#0MS;
   S704_LM_DC_2ND_CLAMP3.Error_T2.ATIME := T#0MS;
   S704_LM_DC_2ND_CLAMP3.CHK_Aux1 := FALSE;
   S704_LM_DC_2ND_CLAMP3.CHK_Aux2 := FALSE;
   S704_LM_DC_2ND_CLAMP3.Error_T1_DN := FALSE;
   S704_LM_DC_2ND_CLAMP3.Error_T2_DN := FALSE;
   S704_LM_DC_2ND_CLAMP3.Adv_Memo := FALSE;
   S704_LM_DC_2ND_CLAMP3.Visu_Adv_Arr[0] := FALSE;
   S704_LM_DC_2ND_CLAMP3.Visu_Adv_Arr[1] := FALSE;
   S704_LM_DC_2ND_CLAMP3.Visu_Adv_Arr[2] := FALSE;
   S704_LM_DC_2ND_CLAMP3.Visu_Adv_Arr[3] := FALSE;
   S704_LM_DC_2ND_CLAMP3.Visu_Adv_Arr[4] := FALSE;
   S704_LM_DC_2ND_CLAMP3.Visu_Adv_Arr[5] := FALSE;
   S704_LM_DC_2ND_CLAMP3.Visu_Adv_Arr[6] := FALSE;
   S704_LM_DC_2ND_CLAMP3.Visu_Adv_Arr[7] := FALSE;
   S704_LM_DC_2ND_CLAMP3.Visu_Adv_Arr[8] := FALSE;
   S704_LM_DC_2ND_CLAMP3.Visu_Adv_Arr[9] := FALSE;
   S704_LM_DC_2ND_CLAMP3.Visu_Adv_Arr[10] := FALSE;
   S704_LM_DC_2ND_CLAMP3.Visu_Adv_Arr[11] := FALSE;
   S704_LM_DC_2ND_CLAMP3.Visu_Adv_Arr[12] := FALSE;
   S704_LM_DC_2ND_CLAMP3.Visu_Adv_Arr[13] := FALSE;
   S704_LM_DC_2ND_CLAMP3.Visu_Adv_Arr[14] := FALSE;
   S704_LM_DC_2ND_CLAMP3.Visu_Adv_Arr[15] := FALSE;
   S704_LM_DC_2ND_CLAMP3.Visu_Ret_Arr[0] := FALSE;
   S704_LM_DC_2ND_CLAMP3.Visu_Ret_Arr[1] := FALSE;
   S704_LM_DC_2ND_CLAMP3.Visu_Ret_Arr[2] := FALSE;
   S704_LM_DC_2ND_CLAMP3.Visu_Ret_Arr[3] := FALSE;
   S704_LM_DC_2ND_CLAMP3.Visu_Ret_Arr[4] := FALSE;
   S704_LM_DC_2ND_CLAMP3.Visu_Ret_Arr[5] := FALSE;
   S704_LM_DC_2ND_CLAMP3.Visu_Ret_Arr[6] := FALSE;
   S704_LM_DC_2ND_CLAMP3.Visu_Ret_Arr[7] := FALSE;
   S704_LM_DC_2ND_CLAMP3.Visu_Ret_Arr[8] := FALSE;
   S704_LM_DC_2ND_CLAMP3.Visu_Ret_Arr[9] := FALSE;
   S704_LM_DC_2ND_CLAMP3.Visu_Ret_Arr[10] := FALSE;
   S704_LM_DC_2ND_CLAMP3.Visu_Ret_Arr[11] := FALSE;
   S704_LM_DC_2ND_CLAMP3.Visu_Ret_Arr[12] := FALSE;
   S704_LM_DC_2ND_CLAMP3.Visu_Ret_Arr[13] := FALSE;
   S704_LM_DC_2ND_CLAMP3.Visu_Ret_Arr[14] := FALSE;
   S704_LM_DC_2ND_CLAMP3.Visu_Ret_Arr[15] := FALSE;
   S704_LM_DC_2ND_CLAMP3.BLK_Move_Ret := 0;
   S704_LM_DC_2ND_CLAMP3.Enable := FALSE;
   S704_LM_DC_2ND_CLAMP3.Adv_End := FALSE;
   S704_LM_DC_2ND_CLAMP3.Ret_End := FALSE;
   S704_LM_DC_2ND_CLAMP4.Enable_Aux := FALSE;
   S704_LM_DC_2ND_CLAMP4.Adv_Amount := 0;
   S704_LM_DC_2ND_CLAMP4.Ret_Amount := 0;
   S704_LM_DC_2ND_CLAMP4.LS_Adv1 := FALSE;
   S704_LM_DC_2ND_CLAMP4.LS_Ret1 := FALSE;
   S704_LM_DC_2ND_CLAMP4.LS_Adv2 := FALSE;
   S704_LM_DC_2ND_CLAMP4.LS_Ret2 := FALSE;
   S704_LM_DC_2ND_CLAMP4.LS_Adv3 := FALSE;
   S704_LM_DC_2ND_CLAMP4.LS_Ret3 := FALSE;
   S704_LM_DC_2ND_CLAMP4.LS_Adv4 := FALSE;
   S704_LM_DC_2ND_CLAMP4.LS_Ret4 := FALSE;
   S704_LM_DC_2ND_CLAMP4.SOL_Adv := FALSE;
   S704_LM_DC_2ND_CLAMP4.SOL_Ret := FALSE;
   S704_LM_DC_2ND_CLAMP4.M_Ready := FALSE;
   S704_LM_DC_2ND_CLAMP4.T_CHK1 := T#0MS;
   S704_LM_DC_2ND_CLAMP4.T_CHK2 := T#0MS;
   S704_LM_DC_2ND_CLAMP4.PB_Lamp_CHK := FALSE;
   S704_LM_DC_2ND_CLAMP4.PB_Error_Rst := FALSE;
   S704_LM_DC_2ND_CLAMP4.M_FLICK := FALSE;
   S704_LM_DC_2ND_CLAMP4.M_Adv_Err := FALSE;
   S704_LM_DC_2ND_CLAMP4.M_Ret_Err := FALSE;
   S704_LM_DC_2ND_CLAMP4.LP_Adv := FALSE;
   S704_LM_DC_2ND_CLAMP4.LP_Ret := FALSE;
   S704_LM_DC_2ND_CLAMP4.Visu_Adv := W#16#0;
   S704_LM_DC_2ND_CLAMP4.Visu_Ret := W#16#0;
   S704_LM_DC_2ND_CLAMP4.Error_T1.IN := FALSE;
   S704_LM_DC_2ND_CLAMP4.Error_T1.PT := T#0MS;
   S704_LM_DC_2ND_CLAMP4.Error_T1.Q := FALSE;
   S704_LM_DC_2ND_CLAMP4.Error_T1.ET := T#0MS;
   S704_LM_DC_2ND_CLAMP4.Error_T1.STATE := B#16#0;
   S704_LM_DC_2ND_CLAMP4.Error_T1.STIME := T#0MS;
   S704_LM_DC_2ND_CLAMP4.Error_T1.ATIME := T#0MS;
   S704_LM_DC_2ND_CLAMP4.Error_T2.IN := FALSE;
   S704_LM_DC_2ND_CLAMP4.Error_T2.PT := T#0MS;
   S704_LM_DC_2ND_CLAMP4.Error_T2.Q := FALSE;
   S704_LM_DC_2ND_CLAMP4.Error_T2.ET := T#0MS;
   S704_LM_DC_2ND_CLAMP4.Error_T2.STATE := B#16#0;
   S704_LM_DC_2ND_CLAMP4.Error_T2.STIME := T#0MS;
   S704_LM_DC_2ND_CLAMP4.Error_T2.ATIME := T#0MS;
   S704_LM_DC_2ND_CLAMP4.CHK_Aux1 := FALSE;
   S704_LM_DC_2ND_CLAMP4.CHK_Aux2 := FALSE;
   S704_LM_DC_2ND_CLAMP4.Error_T1_DN := FALSE;
   S704_LM_DC_2ND_CLAMP4.Error_T2_DN := FALSE;
   S704_LM_DC_2ND_CLAMP4.Adv_Memo := FALSE;
   S704_LM_DC_2ND_CLAMP4.Visu_Adv_Arr[0] := FALSE;
   S704_LM_DC_2ND_CLAMP4.Visu_Adv_Arr[1] := FALSE;
   S704_LM_DC_2ND_CLAMP4.Visu_Adv_Arr[2] := FALSE;
   S704_LM_DC_2ND_CLAMP4.Visu_Adv_Arr[3] := FALSE;
   S704_LM_DC_2ND_CLAMP4.Visu_Adv_Arr[4] := FALSE;
   S704_LM_DC_2ND_CLAMP4.Visu_Adv_Arr[5] := FALSE;
   S704_LM_DC_2ND_CLAMP4.Visu_Adv_Arr[6] := FALSE;
   S704_LM_DC_2ND_CLAMP4.Visu_Adv_Arr[7] := FALSE;
   S704_LM_DC_2ND_CLAMP4.Visu_Adv_Arr[8] := FALSE;
   S704_LM_DC_2ND_CLAMP4.Visu_Adv_Arr[9] := FALSE;
   S704_LM_DC_2ND_CLAMP4.Visu_Adv_Arr[10] := FALSE;
   S704_LM_DC_2ND_CLAMP4.Visu_Adv_Arr[11] := FALSE;
   S704_LM_DC_2ND_CLAMP4.Visu_Adv_Arr[12] := FALSE;
   S704_LM_DC_2ND_CLAMP4.Visu_Adv_Arr[13] := FALSE;
   S704_LM_DC_2ND_CLAMP4.Visu_Adv_Arr[14] := FALSE;
   S704_LM_DC_2ND_CLAMP4.Visu_Adv_Arr[15] := FALSE;
   S704_LM_DC_2ND_CLAMP4.Visu_Ret_Arr[0] := FALSE;
   S704_LM_DC_2ND_CLAMP4.Visu_Ret_Arr[1] := FALSE;
   S704_LM_DC_2ND_CLAMP4.Visu_Ret_Arr[2] := FALSE;
   S704_LM_DC_2ND_CLAMP4.Visu_Ret_Arr[3] := FALSE;
   S704_LM_DC_2ND_CLAMP4.Visu_Ret_Arr[4] := FALSE;
   S704_LM_DC_2ND_CLAMP4.Visu_Ret_Arr[5] := FALSE;
   S704_LM_DC_2ND_CLAMP4.Visu_Ret_Arr[6] := FALSE;
   S704_LM_DC_2ND_CLAMP4.Visu_Ret_Arr[7] := FALSE;
   S704_LM_DC_2ND_CLAMP4.Visu_Ret_Arr[8] := FALSE;
   S704_LM_DC_2ND_CLAMP4.Visu_Ret_Arr[9] := FALSE;
   S704_LM_DC_2ND_CLAMP4.Visu_Ret_Arr[10] := FALSE;
   S704_LM_DC_2ND_CLAMP4.Visu_Ret_Arr[11] := FALSE;
   S704_LM_DC_2ND_CLAMP4.Visu_Ret_Arr[12] := FALSE;
   S704_LM_DC_2ND_CLAMP4.Visu_Ret_Arr[13] := FALSE;
   S704_LM_DC_2ND_CLAMP4.Visu_Ret_Arr[14] := FALSE;
   S704_LM_DC_2ND_CLAMP4.Visu_Ret_Arr[15] := FALSE;
   S704_LM_DC_2ND_CLAMP4.BLK_Move_Ret := 0;
   S704_LM_DC_2ND_CLAMP4.Enable := FALSE;
   S704_LM_DC_2ND_CLAMP4.Adv_End := FALSE;
   S704_LM_DC_2ND_CLAMP4.Ret_End := FALSE;
   S704_LM_DC_2ND_CLAMP5.Enable_Aux := FALSE;
   S704_LM_DC_2ND_CLAMP5.Adv_Amount := 0;
   S704_LM_DC_2ND_CLAMP5.Ret_Amount := 0;
   S704_LM_DC_2ND_CLAMP5.LS_Adv1 := FALSE;
   S704_LM_DC_2ND_CLAMP5.LS_Ret1 := FALSE;
   S704_LM_DC_2ND_CLAMP5.LS_Adv2 := FALSE;
   S704_LM_DC_2ND_CLAMP5.LS_Ret2 := FALSE;
   S704_LM_DC_2ND_CLAMP5.LS_Adv3 := FALSE;
   S704_LM_DC_2ND_CLAMP5.LS_Ret3 := FALSE;
   S704_LM_DC_2ND_CLAMP5.LS_Adv4 := FALSE;
   S704_LM_DC_2ND_CLAMP5.LS_Ret4 := FALSE;
   S704_LM_DC_2ND_CLAMP5.SOL_Adv := FALSE;
   S704_LM_DC_2ND_CLAMP5.SOL_Ret := FALSE;
   S704_LM_DC_2ND_CLAMP5.M_Ready := FALSE;
   S704_LM_DC_2ND_CLAMP5.T_CHK1 := T#0MS;
   S704_LM_DC_2ND_CLAMP5.T_CHK2 := T#0MS;
   S704_LM_DC_2ND_CLAMP5.PB_Lamp_CHK := FALSE;
   S704_LM_DC_2ND_CLAMP5.PB_Error_Rst := FALSE;
   S704_LM_DC_2ND_CLAMP5.M_FLICK := FALSE;
   S704_LM_DC_2ND_CLAMP5.M_Adv_Err := FALSE;
   S704_LM_DC_2ND_CLAMP5.M_Ret_Err := FALSE;
   S704_LM_DC_2ND_CLAMP5.LP_Adv := FALSE;
   S704_LM_DC_2ND_CLAMP5.LP_Ret := FALSE;
   S704_LM_DC_2ND_CLAMP5.Visu_Adv := W#16#0;
   S704_LM_DC_2ND_CLAMP5.Visu_Ret := W#16#0;
   S704_LM_DC_2ND_CLAMP5.Error_T1.IN := FALSE;
   S704_LM_DC_2ND_CLAMP5.Error_T1.PT := T#0MS;
   S704_LM_DC_2ND_CLAMP5.Error_T1.Q := FALSE;
   S704_LM_DC_2ND_CLAMP5.Error_T1.ET := T#0MS;
   S704_LM_DC_2ND_CLAMP5.Error_T1.STATE := B#16#0;
   S704_LM_DC_2ND_CLAMP5.Error_T1.STIME := T#0MS;
   S704_LM_DC_2ND_CLAMP5.Error_T1.ATIME := T#0MS;
   S704_LM_DC_2ND_CLAMP5.Error_T2.IN := FALSE;
   S704_LM_DC_2ND_CLAMP5.Error_T2.PT := T#0MS;
   S704_LM_DC_2ND_CLAMP5.Error_T2.Q := FALSE;
   S704_LM_DC_2ND_CLAMP5.Error_T2.ET := T#0MS;
   S704_LM_DC_2ND_CLAMP5.Error_T2.STATE := B#16#0;
   S704_LM_DC_2ND_CLAMP5.Error_T2.STIME := T#0MS;
   S704_LM_DC_2ND_CLAMP5.Error_T2.ATIME := T#0MS;
   S704_LM_DC_2ND_CLAMP5.CHK_Aux1 := FALSE;
   S704_LM_DC_2ND_CLAMP5.CHK_Aux2 := FALSE;
   S704_LM_DC_2ND_CLAMP5.Error_T1_DN := FALSE;
   S704_LM_DC_2ND_CLAMP5.Error_T2_DN := FALSE;
   S704_LM_DC_2ND_CLAMP5.Adv_Memo := FALSE;
   S704_LM_DC_2ND_CLAMP5.Visu_Adv_Arr[0] := FALSE;
   S704_LM_DC_2ND_CLAMP5.Visu_Adv_Arr[1] := FALSE;
   S704_LM_DC_2ND_CLAMP5.Visu_Adv_Arr[2] := FALSE;
   S704_LM_DC_2ND_CLAMP5.Visu_Adv_Arr[3] := FALSE;
   S704_LM_DC_2ND_CLAMP5.Visu_Adv_Arr[4] := FALSE;
   S704_LM_DC_2ND_CLAMP5.Visu_Adv_Arr[5] := FALSE;
   S704_LM_DC_2ND_CLAMP5.Visu_Adv_Arr[6] := FALSE;
   S704_LM_DC_2ND_CLAMP5.Visu_Adv_Arr[7] := FALSE;
   S704_LM_DC_2ND_CLAMP5.Visu_Adv_Arr[8] := FALSE;
   S704_LM_DC_2ND_CLAMP5.Visu_Adv_Arr[9] := FALSE;
   S704_LM_DC_2ND_CLAMP5.Visu_Adv_Arr[10] := FALSE;
   S704_LM_DC_2ND_CLAMP5.Visu_Adv_Arr[11] := FALSE;
   S704_LM_DC_2ND_CLAMP5.Visu_Adv_Arr[12] := FALSE;
   S704_LM_DC_2ND_CLAMP5.Visu_Adv_Arr[13] := FALSE;
   S704_LM_DC_2ND_CLAMP5.Visu_Adv_Arr[14] := FALSE;
   S704_LM_DC_2ND_CLAMP5.Visu_Adv_Arr[15] := FALSE;
   S704_LM_DC_2ND_CLAMP5.Visu_Ret_Arr[0] := FALSE;
   S704_LM_DC_2ND_CLAMP5.Visu_Ret_Arr[1] := FALSE;
   S704_LM_DC_2ND_CLAMP5.Visu_Ret_Arr[2] := FALSE;
   S704_LM_DC_2ND_CLAMP5.Visu_Ret_Arr[3] := FALSE;
   S704_LM_DC_2ND_CLAMP5.Visu_Ret_Arr[4] := FALSE;
   S704_LM_DC_2ND_CLAMP5.Visu_Ret_Arr[5] := FALSE;
   S704_LM_DC_2ND_CLAMP5.Visu_Ret_Arr[6] := FALSE;
   S704_LM_DC_2ND_CLAMP5.Visu_Ret_Arr[7] := FALSE;
   S704_LM_DC_2ND_CLAMP5.Visu_Ret_Arr[8] := FALSE;
   S704_LM_DC_2ND_CLAMP5.Visu_Ret_Arr[9] := FALSE;
   S704_LM_DC_2ND_CLAMP5.Visu_Ret_Arr[10] := FALSE;
   S704_LM_DC_2ND_CLAMP5.Visu_Ret_Arr[11] := FALSE;
   S704_LM_DC_2ND_CLAMP5.Visu_Ret_Arr[12] := FALSE;
   S704_LM_DC_2ND_CLAMP5.Visu_Ret_Arr[13] := FALSE;
   S704_LM_DC_2ND_CLAMP5.Visu_Ret_Arr[14] := FALSE;
   S704_LM_DC_2ND_CLAMP5.Visu_Ret_Arr[15] := FALSE;
   S704_LM_DC_2ND_CLAMP5.BLK_Move_Ret := 0;
   S704_LM_DC_2ND_CLAMP5.Enable := FALSE;
   S704_LM_DC_2ND_CLAMP5.Adv_End := FALSE;
   S704_LM_DC_2ND_CLAMP5.Ret_End := FALSE;
   S704_LM_DC_STK_PIN.Enable_Aux := FALSE;
   S704_LM_DC_STK_PIN.Adv_Amount := 0;
   S704_LM_DC_STK_PIN.Ret_Amount := 0;
   S704_LM_DC_STK_PIN.LS_Adv1 := FALSE;
   S704_LM_DC_STK_PIN.LS_Ret1 := FALSE;
   S704_LM_DC_STK_PIN.LS_Adv2 := FALSE;
   S704_LM_DC_STK_PIN.LS_Ret2 := FALSE;
   S704_LM_DC_STK_PIN.LS_Adv3 := FALSE;
   S704_LM_DC_STK_PIN.LS_Ret3 := FALSE;
   S704_LM_DC_STK_PIN.LS_Adv4 := FALSE;
   S704_LM_DC_STK_PIN.LS_Ret4 := FALSE;
   S704_LM_DC_STK_PIN.SOL_Adv := FALSE;
   S704_LM_DC_STK_PIN.SOL_Ret := FALSE;
   S704_LM_DC_STK_PIN.M_Ready := FALSE;
   S704_LM_DC_STK_PIN.T_CHK1 := T#0MS;
   S704_LM_DC_STK_PIN.T_CHK2 := T#0MS;
   S704_LM_DC_STK_PIN.PB_Lamp_CHK := FALSE;
   S704_LM_DC_STK_PIN.PB_Error_Rst := FALSE;
   S704_LM_DC_STK_PIN.M_FLICK := FALSE;
   S704_LM_DC_STK_PIN.M_Adv_Err := FALSE;
   S704_LM_DC_STK_PIN.M_Ret_Err := FALSE;
   S704_LM_DC_STK_PIN.LP_Adv := FALSE;
   S704_LM_DC_STK_PIN.LP_Ret := FALSE;
   S704_LM_DC_STK_PIN.Visu_Adv := W#16#0;
   S704_LM_DC_STK_PIN.Visu_Ret := W#16#0;
   S704_LM_DC_STK_PIN.Error_T1.IN := FALSE;
   S704_LM_DC_STK_PIN.Error_T1.PT := T#0MS;
   S704_LM_DC_STK_PIN.Error_T1.Q := FALSE;
   S704_LM_DC_STK_PIN.Error_T1.ET := T#0MS;
   S704_LM_DC_STK_PIN.Error_T1.STATE := B#16#0;
   S704_LM_DC_STK_PIN.Error_T1.STIME := T#0MS;
   S704_LM_DC_STK_PIN.Error_T1.ATIME := T#0MS;
   S704_LM_DC_STK_PIN.Error_T2.IN := FALSE;
   S704_LM_DC_STK_PIN.Error_T2.PT := T#0MS;
   S704_LM_DC_STK_PIN.Error_T2.Q := FALSE;
   S704_LM_DC_STK_PIN.Error_T2.ET := T#0MS;
   S704_LM_DC_STK_PIN.Error_T2.STATE := B#16#0;
   S704_LM_DC_STK_PIN.Error_T2.STIME := T#0MS;
   S704_LM_DC_STK_PIN.Error_T2.ATIME := T#0MS;
   S704_LM_DC_STK_PIN.CHK_Aux1 := FALSE;
   S704_LM_DC_STK_PIN.CHK_Aux2 := FALSE;
   S704_LM_DC_STK_PIN.Error_T1_DN := FALSE;
   S704_LM_DC_STK_PIN.Error_T2_DN := FALSE;
   S704_LM_DC_STK_PIN.Adv_Memo := FALSE;
   S704_LM_DC_STK_PIN.Visu_Adv_Arr[0] := FALSE;
   S704_LM_DC_STK_PIN.Visu_Adv_Arr[1] := FALSE;
   S704_LM_DC_STK_PIN.Visu_Adv_Arr[2] := FALSE;
   S704_LM_DC_STK_PIN.Visu_Adv_Arr[3] := FALSE;
   S704_LM_DC_STK_PIN.Visu_Adv_Arr[4] := FALSE;
   S704_LM_DC_STK_PIN.Visu_Adv_Arr[5] := FALSE;
   S704_LM_DC_STK_PIN.Visu_Adv_Arr[6] := FALSE;
   S704_LM_DC_STK_PIN.Visu_Adv_Arr[7] := FALSE;
   S704_LM_DC_STK_PIN.Visu_Adv_Arr[8] := FALSE;
   S704_LM_DC_STK_PIN.Visu_Adv_Arr[9] := FALSE;
   S704_LM_DC_STK_PIN.Visu_Adv_Arr[10] := FALSE;
   S704_LM_DC_STK_PIN.Visu_Adv_Arr[11] := FALSE;
   S704_LM_DC_STK_PIN.Visu_Adv_Arr[12] := FALSE;
   S704_LM_DC_STK_PIN.Visu_Adv_Arr[13] := FALSE;
   S704_LM_DC_STK_PIN.Visu_Adv_Arr[14] := FALSE;
   S704_LM_DC_STK_PIN.Visu_Adv_Arr[15] := FALSE;
   S704_LM_DC_STK_PIN.Visu_Ret_Arr[0] := FALSE;
   S704_LM_DC_STK_PIN.Visu_Ret_Arr[1] := FALSE;
   S704_LM_DC_STK_PIN.Visu_Ret_Arr[2] := FALSE;
   S704_LM_DC_STK_PIN.Visu_Ret_Arr[3] := FALSE;
   S704_LM_DC_STK_PIN.Visu_Ret_Arr[4] := FALSE;
   S704_LM_DC_STK_PIN.Visu_Ret_Arr[5] := FALSE;
   S704_LM_DC_STK_PIN.Visu_Ret_Arr[6] := FALSE;
   S704_LM_DC_STK_PIN.Visu_Ret_Arr[7] := FALSE;
   S704_LM_DC_STK_PIN.Visu_Ret_Arr[8] := FALSE;
   S704_LM_DC_STK_PIN.Visu_Ret_Arr[9] := FALSE;
   S704_LM_DC_STK_PIN.Visu_Ret_Arr[10] := FALSE;
   S704_LM_DC_STK_PIN.Visu_Ret_Arr[11] := FALSE;
   S704_LM_DC_STK_PIN.Visu_Ret_Arr[12] := FALSE;
   S704_LM_DC_STK_PIN.Visu_Ret_Arr[13] := FALSE;
   S704_LM_DC_STK_PIN.Visu_Ret_Arr[14] := FALSE;
   S704_LM_DC_STK_PIN.Visu_Ret_Arr[15] := FALSE;
   S704_LM_DC_STK_PIN.BLK_Move_Ret := 0;
   S704_LM_DC_STK_PIN.Enable := FALSE;
   S704_LM_DC_STK_PIN.Adv_End := FALSE;
   S704_LM_DC_STK_PIN.Ret_End := FALSE;
   S704_LM_DC_OTR_CLAMP.Enable_Aux := FALSE;
   S704_LM_DC_OTR_CLAMP.Adv_Amount := 0;
   S704_LM_DC_OTR_CLAMP.Ret_Amount := 0;
   S704_LM_DC_OTR_CLAMP.LS_Adv1 := FALSE;
   S704_LM_DC_OTR_CLAMP.LS_Ret1 := FALSE;
   S704_LM_DC_OTR_CLAMP.LS_Adv2 := FALSE;
   S704_LM_DC_OTR_CLAMP.LS_Ret2 := FALSE;
   S704_LM_DC_OTR_CLAMP.LS_Adv3 := FALSE;
   S704_LM_DC_OTR_CLAMP.LS_Ret3 := FALSE;
   S704_LM_DC_OTR_CLAMP.LS_Adv4 := FALSE;
   S704_LM_DC_OTR_CLAMP.LS_Ret4 := FALSE;
   S704_LM_DC_OTR_CLAMP.SOL_Adv := FALSE;
   S704_LM_DC_OTR_CLAMP.SOL_Ret := FALSE;
   S704_LM_DC_OTR_CLAMP.M_Ready := FALSE;
   S704_LM_DC_OTR_CLAMP.T_CHK1 := T#0MS;
   S704_LM_DC_OTR_CLAMP.T_CHK2 := T#0MS;
   S704_LM_DC_OTR_CLAMP.PB_Lamp_CHK := FALSE;
   S704_LM_DC_OTR_CLAMP.PB_Error_Rst := FALSE;
   S704_LM_DC_OTR_CLAMP.M_FLICK := FALSE;
   S704_LM_DC_OTR_CLAMP.M_Adv_Err := FALSE;
   S704_LM_DC_OTR_CLAMP.M_Ret_Err := FALSE;
   S704_LM_DC_OTR_CLAMP.LP_Adv := FALSE;
   S704_LM_DC_OTR_CLAMP.LP_Ret := FALSE;
   S704_LM_DC_OTR_CLAMP.Visu_Adv := W#16#0;
   S704_LM_DC_OTR_CLAMP.Visu_Ret := W#16#0;
   S704_LM_DC_OTR_CLAMP.Error_T1.IN := FALSE;
   S704_LM_DC_OTR_CLAMP.Error_T1.PT := T#0MS;
   S704_LM_DC_OTR_CLAMP.Error_T1.Q := FALSE;
   S704_LM_DC_OTR_CLAMP.Error_T1.ET := T#0MS;
   S704_LM_DC_OTR_CLAMP.Error_T1.STATE := B#16#0;
   S704_LM_DC_OTR_CLAMP.Error_T1.STIME := T#0MS;
   S704_LM_DC_OTR_CLAMP.Error_T1.ATIME := T#0MS;
   S704_LM_DC_OTR_CLAMP.Error_T2.IN := FALSE;
   S704_LM_DC_OTR_CLAMP.Error_T2.PT := T#0MS;
   S704_LM_DC_OTR_CLAMP.Error_T2.Q := FALSE;
   S704_LM_DC_OTR_CLAMP.Error_T2.ET := T#0MS;
   S704_LM_DC_OTR_CLAMP.Error_T2.STATE := B#16#0;
   S704_LM_DC_OTR_CLAMP.Error_T2.STIME := T#0MS;
   S704_LM_DC_OTR_CLAMP.Error_T2.ATIME := T#0MS;
   S704_LM_DC_OTR_CLAMP.CHK_Aux1 := FALSE;
   S704_LM_DC_OTR_CLAMP.CHK_Aux2 := FALSE;
   S704_LM_DC_OTR_CLAMP.Error_T1_DN := FALSE;
   S704_LM_DC_OTR_CLAMP.Error_T2_DN := FALSE;
   S704_LM_DC_OTR_CLAMP.Adv_Memo := FALSE;
   S704_LM_DC_OTR_CLAMP.Visu_Adv_Arr[0] := FALSE;
   S704_LM_DC_OTR_CLAMP.Visu_Adv_Arr[1] := FALSE;
   S704_LM_DC_OTR_CLAMP.Visu_Adv_Arr[2] := FALSE;
   S704_LM_DC_OTR_CLAMP.Visu_Adv_Arr[3] := FALSE;
   S704_LM_DC_OTR_CLAMP.Visu_Adv_Arr[4] := FALSE;
   S704_LM_DC_OTR_CLAMP.Visu_Adv_Arr[5] := FALSE;
   S704_LM_DC_OTR_CLAMP.Visu_Adv_Arr[6] := FALSE;
   S704_LM_DC_OTR_CLAMP.Visu_Adv_Arr[7] := FALSE;
   S704_LM_DC_OTR_CLAMP.Visu_Adv_Arr[8] := FALSE;
   S704_LM_DC_OTR_CLAMP.Visu_Adv_Arr[9] := FALSE;
   S704_LM_DC_OTR_CLAMP.Visu_Adv_Arr[10] := FALSE;
   S704_LM_DC_OTR_CLAMP.Visu_Adv_Arr[11] := FALSE;
   S704_LM_DC_OTR_CLAMP.Visu_Adv_Arr[12] := FALSE;
   S704_LM_DC_OTR_CLAMP.Visu_Adv_Arr[13] := FALSE;
   S704_LM_DC_OTR_CLAMP.Visu_Adv_Arr[14] := FALSE;
   S704_LM_DC_OTR_CLAMP.Visu_Adv_Arr[15] := FALSE;
   S704_LM_DC_OTR_CLAMP.Visu_Ret_Arr[0] := FALSE;
   S704_LM_DC_OTR_CLAMP.Visu_Ret_Arr[1] := FALSE;
   S704_LM_DC_OTR_CLAMP.Visu_Ret_Arr[2] := FALSE;
   S704_LM_DC_OTR_CLAMP.Visu_Ret_Arr[3] := FALSE;
   S704_LM_DC_OTR_CLAMP.Visu_Ret_Arr[4] := FALSE;
   S704_LM_DC_OTR_CLAMP.Visu_Ret_Arr[5] := FALSE;
   S704_LM_DC_OTR_CLAMP.Visu_Ret_Arr[6] := FALSE;
   S704_LM_DC_OTR_CLAMP.Visu_Ret_Arr[7] := FALSE;
   S704_LM_DC_OTR_CLAMP.Visu_Ret_Arr[8] := FALSE;
   S704_LM_DC_OTR_CLAMP.Visu_Ret_Arr[9] := FALSE;
   S704_LM_DC_OTR_CLAMP.Visu_Ret_Arr[10] := FALSE;
   S704_LM_DC_OTR_CLAMP.Visu_Ret_Arr[11] := FALSE;
   S704_LM_DC_OTR_CLAMP.Visu_Ret_Arr[12] := FALSE;
   S704_LM_DC_OTR_CLAMP.Visu_Ret_Arr[13] := FALSE;
   S704_LM_DC_OTR_CLAMP.Visu_Ret_Arr[14] := FALSE;
   S704_LM_DC_OTR_CLAMP.Visu_Ret_Arr[15] := FALSE;
   S704_LM_DC_OTR_CLAMP.BLK_Move_Ret := 0;
   S704_LM_DC_OTR_CLAMP.Enable := FALSE;
   S704_LM_DC_OTR_CLAMP.Adv_End := FALSE;
   S704_LM_DC_OTR_CLAMP.Ret_End := FALSE;
   S704_LM_DC_ASSY_CLAMP.Enable_Aux := FALSE;
   S704_LM_DC_ASSY_CLAMP.Adv_Amount := 0;
   S704_LM_DC_ASSY_CLAMP.Ret_Amount := 0;
   S704_LM_DC_ASSY_CLAMP.LS_Adv1 := FALSE;
   S704_LM_DC_ASSY_CLAMP.LS_Ret1 := FALSE;
   S704_LM_DC_ASSY_CLAMP.LS_Adv2 := FALSE;
   S704_LM_DC_ASSY_CLAMP.LS_Ret2 := FALSE;
   S704_LM_DC_ASSY_CLAMP.LS_Adv3 := FALSE;
   S704_LM_DC_ASSY_CLAMP.LS_Ret3 := FALSE;
   S704_LM_DC_ASSY_CLAMP.LS_Adv4 := FALSE;
   S704_LM_DC_ASSY_CLAMP.LS_Ret4 := FALSE;
   S704_LM_DC_ASSY_CLAMP.SOL_Adv := FALSE;
   S704_LM_DC_ASSY_CLAMP.SOL_Ret := FALSE;
   S704_LM_DC_ASSY_CLAMP.M_Ready := FALSE;
   S704_LM_DC_ASSY_CLAMP.T_CHK1 := T#0MS;
   S704_LM_DC_ASSY_CLAMP.T_CHK2 := T#0MS;
   S704_LM_DC_ASSY_CLAMP.PB_Lamp_CHK := FALSE;
   S704_LM_DC_ASSY_CLAMP.PB_Error_Rst := FALSE;
   S704_LM_DC_ASSY_CLAMP.M_FLICK := FALSE;
   S704_LM_DC_ASSY_CLAMP.M_Adv_Err := FALSE;
   S704_LM_DC_ASSY_CLAMP.M_Ret_Err := FALSE;
   S704_LM_DC_ASSY_CLAMP.LP_Adv := FALSE;
   S704_LM_DC_ASSY_CLAMP.LP_Ret := FALSE;
   S704_LM_DC_ASSY_CLAMP.Visu_Adv := W#16#0;
   S704_LM_DC_ASSY_CLAMP.Visu_Ret := W#16#0;
   S704_LM_DC_ASSY_CLAMP.Error_T1.IN := FALSE;
   S704_LM_DC_ASSY_CLAMP.Error_T1.PT := T#0MS;
   S704_LM_DC_ASSY_CLAMP.Error_T1.Q := FALSE;
   S704_LM_DC_ASSY_CLAMP.Error_T1.ET := T#0MS;
   S704_LM_DC_ASSY_CLAMP.Error_T1.STATE := B#16#0;
   S704_LM_DC_ASSY_CLAMP.Error_T1.STIME := T#0MS;
   S704_LM_DC_ASSY_CLAMP.Error_T1.ATIME := T#0MS;
   S704_LM_DC_ASSY_CLAMP.Error_T2.IN := FALSE;
   S704_LM_DC_ASSY_CLAMP.Error_T2.PT := T#0MS;
   S704_LM_DC_ASSY_CLAMP.Error_T2.Q := FALSE;
   S704_LM_DC_ASSY_CLAMP.Error_T2.ET := T#0MS;
   S704_LM_DC_ASSY_CLAMP.Error_T2.STATE := B#16#0;
   S704_LM_DC_ASSY_CLAMP.Error_T2.STIME := T#0MS;
   S704_LM_DC_ASSY_CLAMP.Error_T2.ATIME := T#0MS;
   S704_LM_DC_ASSY_CLAMP.CHK_Aux1 := FALSE;
   S704_LM_DC_ASSY_CLAMP.CHK_Aux2 := FALSE;
   S704_LM_DC_ASSY_CLAMP.Error_T1_DN := FALSE;
   S704_LM_DC_ASSY_CLAMP.Error_T2_DN := FALSE;
   S704_LM_DC_ASSY_CLAMP.Adv_Memo := FALSE;
   S704_LM_DC_ASSY_CLAMP.Visu_Adv_Arr[0] := FALSE;
   S704_LM_DC_ASSY_CLAMP.Visu_Adv_Arr[1] := FALSE;
   S704_LM_DC_ASSY_CLAMP.Visu_Adv_Arr[2] := FALSE;
   S704_LM_DC_ASSY_CLAMP.Visu_Adv_Arr[3] := FALSE;
   S704_LM_DC_ASSY_CLAMP.Visu_Adv_Arr[4] := FALSE;
   S704_LM_DC_ASSY_CLAMP.Visu_Adv_Arr[5] := FALSE;
   S704_LM_DC_ASSY_CLAMP.Visu_Adv_Arr[6] := FALSE;
   S704_LM_DC_ASSY_CLAMP.Visu_Adv_Arr[7] := FALSE;
   S704_LM_DC_ASSY_CLAMP.Visu_Adv_Arr[8] := FALSE;
   S704_LM_DC_ASSY_CLAMP.Visu_Adv_Arr[9] := FALSE;
   S704_LM_DC_ASSY_CLAMP.Visu_Adv_Arr[10] := FALSE;
   S704_LM_DC_ASSY_CLAMP.Visu_Adv_Arr[11] := FALSE;
   S704_LM_DC_ASSY_CLAMP.Visu_Adv_Arr[12] := FALSE;
   S704_LM_DC_ASSY_CLAMP.Visu_Adv_Arr[13] := FALSE;
   S704_LM_DC_ASSY_CLAMP.Visu_Adv_Arr[14] := FALSE;
   S704_LM_DC_ASSY_CLAMP.Visu_Adv_Arr[15] := FALSE;
   S704_LM_DC_ASSY_CLAMP.Visu_Ret_Arr[0] := FALSE;
   S704_LM_DC_ASSY_CLAMP.Visu_Ret_Arr[1] := FALSE;
   S704_LM_DC_ASSY_CLAMP.Visu_Ret_Arr[2] := FALSE;
   S704_LM_DC_ASSY_CLAMP.Visu_Ret_Arr[3] := FALSE;
   S704_LM_DC_ASSY_CLAMP.Visu_Ret_Arr[4] := FALSE;
   S704_LM_DC_ASSY_CLAMP.Visu_Ret_Arr[5] := FALSE;
   S704_LM_DC_ASSY_CLAMP.Visu_Ret_Arr[6] := FALSE;
   S704_LM_DC_ASSY_CLAMP.Visu_Ret_Arr[7] := FALSE;
   S704_LM_DC_ASSY_CLAMP.Visu_Ret_Arr[8] := FALSE;
   S704_LM_DC_ASSY_CLAMP.Visu_Ret_Arr[9] := FALSE;
   S704_LM_DC_ASSY_CLAMP.Visu_Ret_Arr[10] := FALSE;
   S704_LM_DC_ASSY_CLAMP.Visu_Ret_Arr[11] := FALSE;
   S704_LM_DC_ASSY_CLAMP.Visu_Ret_Arr[12] := FALSE;
   S704_LM_DC_ASSY_CLAMP.Visu_Ret_Arr[13] := FALSE;
   S704_LM_DC_ASSY_CLAMP.Visu_Ret_Arr[14] := FALSE;
   S704_LM_DC_ASSY_CLAMP.Visu_Ret_Arr[15] := FALSE;
   S704_LM_DC_ASSY_CLAMP.BLK_Move_Ret := 0;
   S704_LM_DC_ASSY_CLAMP.Enable := FALSE;
   S704_LM_DC_ASSY_CLAMP.Adv_End := FALSE;
   S704_LM_DC_ASSY_CLAMP.Ret_End := FALSE;
   S704_LM_DC_FF_PIN.Enable_Aux := FALSE;
   S704_LM_DC_FF_PIN.Adv_Amount := 0;
   S704_LM_DC_FF_PIN.Ret_Amount := 0;
   S704_LM_DC_FF_PIN.LS_Adv1 := FALSE;
   S704_LM_DC_FF_PIN.LS_Ret1 := FALSE;
   S704_LM_DC_FF_PIN.LS_Adv2 := FALSE;
   S704_LM_DC_FF_PIN.LS_Ret2 := FALSE;
   S704_LM_DC_FF_PIN.LS_Adv3 := FALSE;
   S704_LM_DC_FF_PIN.LS_Ret3 := FALSE;
   S704_LM_DC_FF_PIN.LS_Adv4 := FALSE;
   S704_LM_DC_FF_PIN.LS_Ret4 := FALSE;
   S704_LM_DC_FF_PIN.SOL_Adv := FALSE;
   S704_LM_DC_FF_PIN.SOL_Ret := FALSE;
   S704_LM_DC_FF_PIN.M_Ready := FALSE;
   S704_LM_DC_FF_PIN.T_CHK1 := T#0MS;
   S704_LM_DC_FF_PIN.T_CHK2 := T#0MS;
   S704_LM_DC_FF_PIN.PB_Lamp_CHK := FALSE;
   S704_LM_DC_FF_PIN.PB_Error_Rst := FALSE;
   S704_LM_DC_FF_PIN.M_FLICK := FALSE;
   S704_LM_DC_FF_PIN.M_Adv_Err := FALSE;
   S704_LM_DC_FF_PIN.M_Ret_Err := FALSE;
   S704_LM_DC_FF_PIN.LP_Adv := FALSE;
   S704_LM_DC_FF_PIN.LP_Ret := FALSE;
   S704_LM_DC_FF_PIN.Visu_Adv := W#16#0;
   S704_LM_DC_FF_PIN.Visu_Ret := W#16#0;
   S704_LM_DC_FF_PIN.Error_T1.IN := FALSE;
   S704_LM_DC_FF_PIN.Error_T1.PT := T#0MS;
   S704_LM_DC_FF_PIN.Error_T1.Q := FALSE;
   S704_LM_DC_FF_PIN.Error_T1.ET := T#0MS;
   S704_LM_DC_FF_PIN.Error_T1.STATE := B#16#0;
   S704_LM_DC_FF_PIN.Error_T1.STIME := T#0MS;
   S704_LM_DC_FF_PIN.Error_T1.ATIME := T#0MS;
   S704_LM_DC_FF_PIN.Error_T2.IN := FALSE;
   S704_LM_DC_FF_PIN.Error_T2.PT := T#0MS;
   S704_LM_DC_FF_PIN.Error_T2.Q := FALSE;
   S704_LM_DC_FF_PIN.Error_T2.ET := T#0MS;
   S704_LM_DC_FF_PIN.Error_T2.STATE := B#16#0;
   S704_LM_DC_FF_PIN.Error_T2.STIME := T#0MS;
   S704_LM_DC_FF_PIN.Error_T2.ATIME := T#0MS;
   S704_LM_DC_FF_PIN.CHK_Aux1 := FALSE;
   S704_LM_DC_FF_PIN.CHK_Aux2 := FALSE;
   S704_LM_DC_FF_PIN.Error_T1_DN := FALSE;
   S704_LM_DC_FF_PIN.Error_T2_DN := FALSE;
   S704_LM_DC_FF_PIN.Adv_Memo := FALSE;
   S704_LM_DC_FF_PIN.Visu_Adv_Arr[0] := FALSE;
   S704_LM_DC_FF_PIN.Visu_Adv_Arr[1] := FALSE;
   S704_LM_DC_FF_PIN.Visu_Adv_Arr[2] := FALSE;
   S704_LM_DC_FF_PIN.Visu_Adv_Arr[3] := FALSE;
   S704_LM_DC_FF_PIN.Visu_Adv_Arr[4] := FALSE;
   S704_LM_DC_FF_PIN.Visu_Adv_Arr[5] := FALSE;
   S704_LM_DC_FF_PIN.Visu_Adv_Arr[6] := FALSE;
   S704_LM_DC_FF_PIN.Visu_Adv_Arr[7] := FALSE;
   S704_LM_DC_FF_PIN.Visu_Adv_Arr[8] := FALSE;
   S704_LM_DC_FF_PIN.Visu_Adv_Arr[9] := FALSE;
   S704_LM_DC_FF_PIN.Visu_Adv_Arr[10] := FALSE;
   S704_LM_DC_FF_PIN.Visu_Adv_Arr[11] := FALSE;
   S704_LM_DC_FF_PIN.Visu_Adv_Arr[12] := FALSE;
   S704_LM_DC_FF_PIN.Visu_Adv_Arr[13] := FALSE;
   S704_LM_DC_FF_PIN.Visu_Adv_Arr[14] := FALSE;
   S704_LM_DC_FF_PIN.Visu_Adv_Arr[15] := FALSE;
   S704_LM_DC_FF_PIN.Visu_Ret_Arr[0] := FALSE;
   S704_LM_DC_FF_PIN.Visu_Ret_Arr[1] := FALSE;
   S704_LM_DC_FF_PIN.Visu_Ret_Arr[2] := FALSE;
   S704_LM_DC_FF_PIN.Visu_Ret_Arr[3] := FALSE;
   S704_LM_DC_FF_PIN.Visu_Ret_Arr[4] := FALSE;
   S704_LM_DC_FF_PIN.Visu_Ret_Arr[5] := FALSE;
   S704_LM_DC_FF_PIN.Visu_Ret_Arr[6] := FALSE;
   S704_LM_DC_FF_PIN.Visu_Ret_Arr[7] := FALSE;
   S704_LM_DC_FF_PIN.Visu_Ret_Arr[8] := FALSE;
   S704_LM_DC_FF_PIN.Visu_Ret_Arr[9] := FALSE;
   S704_LM_DC_FF_PIN.Visu_Ret_Arr[10] := FALSE;
   S704_LM_DC_FF_PIN.Visu_Ret_Arr[11] := FALSE;
   S704_LM_DC_FF_PIN.Visu_Ret_Arr[12] := FALSE;
   S704_LM_DC_FF_PIN.Visu_Ret_Arr[13] := FALSE;
   S704_LM_DC_FF_PIN.Visu_Ret_Arr[14] := FALSE;
   S704_LM_DC_FF_PIN.Visu_Ret_Arr[15] := FALSE;
   S704_LM_DC_FF_PIN.BLK_Move_Ret := 0;
   S704_LM_DC_FF_PIN.Enable := FALSE;
   S704_LM_DC_FF_PIN.Adv_End := FALSE;
   S704_LM_DC_FF_PIN.Ret_End := FALSE;
   S704_LM_DC_FF_CLAMP.Enable_Aux := FALSE;
   S704_LM_DC_FF_CLAMP.Adv_Amount := 0;
   S704_LM_DC_FF_CLAMP.Ret_Amount := 0;
   S704_LM_DC_FF_CLAMP.LS_Adv1 := FALSE;
   S704_LM_DC_FF_CLAMP.LS_Ret1 := FALSE;
   S704_LM_DC_FF_CLAMP.LS_Adv2 := FALSE;
   S704_LM_DC_FF_CLAMP.LS_Ret2 := FALSE;
   S704_LM_DC_FF_CLAMP.LS_Adv3 := FALSE;
   S704_LM_DC_FF_CLAMP.LS_Ret3 := FALSE;
   S704_LM_DC_FF_CLAMP.LS_Adv4 := FALSE;
   S704_LM_DC_FF_CLAMP.LS_Ret4 := FALSE;
   S704_LM_DC_FF_CLAMP.SOL_Adv := FALSE;
   S704_LM_DC_FF_CLAMP.SOL_Ret := FALSE;
   S704_LM_DC_FF_CLAMP.M_Ready := FALSE;
   S704_LM_DC_FF_CLAMP.T_CHK1 := T#0MS;
   S704_LM_DC_FF_CLAMP.T_CHK2 := T#0MS;
   S704_LM_DC_FF_CLAMP.PB_Lamp_CHK := FALSE;
   S704_LM_DC_FF_CLAMP.PB_Error_Rst := FALSE;
   S704_LM_DC_FF_CLAMP.M_FLICK := FALSE;
   S704_LM_DC_FF_CLAMP.M_Adv_Err := FALSE;
   S704_LM_DC_FF_CLAMP.M_Ret_Err := FALSE;
   S704_LM_DC_FF_CLAMP.LP_Adv := FALSE;
   S704_LM_DC_FF_CLAMP.LP_Ret := FALSE;
   S704_LM_DC_FF_CLAMP.Visu_Adv := W#16#0;
   S704_LM_DC_FF_CLAMP.Visu_Ret := W#16#0;
   S704_LM_DC_FF_CLAMP.Error_T1.IN := FALSE;
   S704_LM_DC_FF_CLAMP.Error_T1.PT := T#0MS;
   S704_LM_DC_FF_CLAMP.Error_T1.Q := FALSE;
   S704_LM_DC_FF_CLAMP.Error_T1.ET := T#0MS;
   S704_LM_DC_FF_CLAMP.Error_T1.STATE := B#16#0;
   S704_LM_DC_FF_CLAMP.Error_T1.STIME := T#0MS;
   S704_LM_DC_FF_CLAMP.Error_T1.ATIME := T#0MS;
   S704_LM_DC_FF_CLAMP.Error_T2.IN := FALSE;
   S704_LM_DC_FF_CLAMP.Error_T2.PT := T#0MS;
   S704_LM_DC_FF_CLAMP.Error_T2.Q := FALSE;
   S704_LM_DC_FF_CLAMP.Error_T2.ET := T#0MS;
   S704_LM_DC_FF_CLAMP.Error_T2.STATE := B#16#0;
   S704_LM_DC_FF_CLAMP.Error_T2.STIME := T#0MS;
   S704_LM_DC_FF_CLAMP.Error_T2.ATIME := T#0MS;
   S704_LM_DC_FF_CLAMP.CHK_Aux1 := FALSE;
   S704_LM_DC_FF_CLAMP.CHK_Aux2 := FALSE;
   S704_LM_DC_FF_CLAMP.Error_T1_DN := FALSE;
   S704_LM_DC_FF_CLAMP.Error_T2_DN := FALSE;
   S704_LM_DC_FF_CLAMP.Adv_Memo := FALSE;
   S704_LM_DC_FF_CLAMP.Visu_Adv_Arr[0] := FALSE;
   S704_LM_DC_FF_CLAMP.Visu_Adv_Arr[1] := FALSE;
   S704_LM_DC_FF_CLAMP.Visu_Adv_Arr[2] := FALSE;
   S704_LM_DC_FF_CLAMP.Visu_Adv_Arr[3] := FALSE;
   S704_LM_DC_FF_CLAMP.Visu_Adv_Arr[4] := FALSE;
   S704_LM_DC_FF_CLAMP.Visu_Adv_Arr[5] := FALSE;
   S704_LM_DC_FF_CLAMP.Visu_Adv_Arr[6] := FALSE;
   S704_LM_DC_FF_CLAMP.Visu_Adv_Arr[7] := FALSE;
   S704_LM_DC_FF_CLAMP.Visu_Adv_Arr[8] := FALSE;
   S704_LM_DC_FF_CLAMP.Visu_Adv_Arr[9] := FALSE;
   S704_LM_DC_FF_CLAMP.Visu_Adv_Arr[10] := FALSE;
   S704_LM_DC_FF_CLAMP.Visu_Adv_Arr[11] := FALSE;
   S704_LM_DC_FF_CLAMP.Visu_Adv_Arr[12] := FALSE;
   S704_LM_DC_FF_CLAMP.Visu_Adv_Arr[13] := FALSE;
   S704_LM_DC_FF_CLAMP.Visu_Adv_Arr[14] := FALSE;
   S704_LM_DC_FF_CLAMP.Visu_Adv_Arr[15] := FALSE;
   S704_LM_DC_FF_CLAMP.Visu_Ret_Arr[0] := FALSE;
   S704_LM_DC_FF_CLAMP.Visu_Ret_Arr[1] := FALSE;
   S704_LM_DC_FF_CLAMP.Visu_Ret_Arr[2] := FALSE;
   S704_LM_DC_FF_CLAMP.Visu_Ret_Arr[3] := FALSE;
   S704_LM_DC_FF_CLAMP.Visu_Ret_Arr[4] := FALSE;
   S704_LM_DC_FF_CLAMP.Visu_Ret_Arr[5] := FALSE;
   S704_LM_DC_FF_CLAMP.Visu_Ret_Arr[6] := FALSE;
   S704_LM_DC_FF_CLAMP.Visu_Ret_Arr[7] := FALSE;
   S704_LM_DC_FF_CLAMP.Visu_Ret_Arr[8] := FALSE;
   S704_LM_DC_FF_CLAMP.Visu_Ret_Arr[9] := FALSE;
   S704_LM_DC_FF_CLAMP.Visu_Ret_Arr[10] := FALSE;
   S704_LM_DC_FF_CLAMP.Visu_Ret_Arr[11] := FALSE;
   S704_LM_DC_FF_CLAMP.Visu_Ret_Arr[12] := FALSE;
   S704_LM_DC_FF_CLAMP.Visu_Ret_Arr[13] := FALSE;
   S704_LM_DC_FF_CLAMP.Visu_Ret_Arr[14] := FALSE;
   S704_LM_DC_FF_CLAMP.Visu_Ret_Arr[15] := FALSE;
   S704_LM_DC_FF_CLAMP.BLK_Move_Ret := 0;
   S704_LM_DC_FF_CLAMP.Enable := FALSE;
   S704_LM_DC_FF_CLAMP.Adv_End := FALSE;
   S704_LM_DC_FF_CLAMP.Ret_End := FALSE;
   S704_LM_DC_2ND_CLAMP6.Enable_Aux := FALSE;
   S704_LM_DC_2ND_CLAMP6.Adv_Amount := 0;
   S704_LM_DC_2ND_CLAMP6.Ret_Amount := 0;
   S704_LM_DC_2ND_CLAMP6.LS_Adv1 := FALSE;
   S704_LM_DC_2ND_CLAMP6.LS_Ret1 := FALSE;
   S704_LM_DC_2ND_CLAMP6.LS_Adv2 := FALSE;
   S704_LM_DC_2ND_CLAMP6.LS_Ret2 := FALSE;
   S704_LM_DC_2ND_CLAMP6.LS_Adv3 := FALSE;
   S704_LM_DC_2ND_CLAMP6.LS_Ret3 := FALSE;
   S704_LM_DC_2ND_CLAMP6.LS_Adv4 := FALSE;
   S704_LM_DC_2ND_CLAMP6.LS_Ret4 := FALSE;
   S704_LM_DC_2ND_CLAMP6.SOL_Adv := FALSE;
   S704_LM_DC_2ND_CLAMP6.SOL_Ret := FALSE;
   S704_LM_DC_2ND_CLAMP6.M_Ready := FALSE;
   S704_LM_DC_2ND_CLAMP6.T_CHK1 := T#0MS;
   S704_LM_DC_2ND_CLAMP6.T_CHK2 := T#0MS;
   S704_LM_DC_2ND_CLAMP6.PB_Lamp_CHK := FALSE;
   S704_LM_DC_2ND_CLAMP6.PB_Error_Rst := FALSE;
   S704_LM_DC_2ND_CLAMP6.M_FLICK := FALSE;
   S704_LM_DC_2ND_CLAMP6.M_Adv_Err := FALSE;
   S704_LM_DC_2ND_CLAMP6.M_Ret_Err := FALSE;
   S704_LM_DC_2ND_CLAMP6.LP_Adv := FALSE;
   S704_LM_DC_2ND_CLAMP6.LP_Ret := FALSE;
   S704_LM_DC_2ND_CLAMP6.Visu_Adv := W#16#0;
   S704_LM_DC_2ND_CLAMP6.Visu_Ret := W#16#0;
   S704_LM_DC_2ND_CLAMP6.Error_T1.IN := FALSE;
   S704_LM_DC_2ND_CLAMP6.Error_T1.PT := T#0MS;
   S704_LM_DC_2ND_CLAMP6.Error_T1.Q := FALSE;
   S704_LM_DC_2ND_CLAMP6.Error_T1.ET := T#0MS;
   S704_LM_DC_2ND_CLAMP6.Error_T1.STATE := B#16#0;
   S704_LM_DC_2ND_CLAMP6.Error_T1.STIME := T#0MS;
   S704_LM_DC_2ND_CLAMP6.Error_T1.ATIME := T#0MS;
   S704_LM_DC_2ND_CLAMP6.Error_T2.IN := FALSE;
   S704_LM_DC_2ND_CLAMP6.Error_T2.PT := T#0MS;
   S704_LM_DC_2ND_CLAMP6.Error_T2.Q := FALSE;
   S704_LM_DC_2ND_CLAMP6.Error_T2.ET := T#0MS;
   S704_LM_DC_2ND_CLAMP6.Error_T2.STATE := B#16#0;
   S704_LM_DC_2ND_CLAMP6.Error_T2.STIME := T#0MS;
   S704_LM_DC_2ND_CLAMP6.Error_T2.ATIME := T#0MS;
   S704_LM_DC_2ND_CLAMP6.CHK_Aux1 := FALSE;
   S704_LM_DC_2ND_CLAMP6.CHK_Aux2 := FALSE;
   S704_LM_DC_2ND_CLAMP6.Error_T1_DN := FALSE;
   S704_LM_DC_2ND_CLAMP6.Error_T2_DN := FALSE;
   S704_LM_DC_2ND_CLAMP6.Adv_Memo := FALSE;
   S704_LM_DC_2ND_CLAMP6.Visu_Adv_Arr[0] := FALSE;
   S704_LM_DC_2ND_CLAMP6.Visu_Adv_Arr[1] := FALSE;
   S704_LM_DC_2ND_CLAMP6.Visu_Adv_Arr[2] := FALSE;
   S704_LM_DC_2ND_CLAMP6.Visu_Adv_Arr[3] := FALSE;
   S704_LM_DC_2ND_CLAMP6.Visu_Adv_Arr[4] := FALSE;
   S704_LM_DC_2ND_CLAMP6.Visu_Adv_Arr[5] := FALSE;
   S704_LM_DC_2ND_CLAMP6.Visu_Adv_Arr[6] := FALSE;
   S704_LM_DC_2ND_CLAMP6.Visu_Adv_Arr[7] := FALSE;
   S704_LM_DC_2ND_CLAMP6.Visu_Adv_Arr[8] := FALSE;
   S704_LM_DC_2ND_CLAMP6.Visu_Adv_Arr[9] := FALSE;
   S704_LM_DC_2ND_CLAMP6.Visu_Adv_Arr[10] := FALSE;
   S704_LM_DC_2ND_CLAMP6.Visu_Adv_Arr[11] := FALSE;
   S704_LM_DC_2ND_CLAMP6.Visu_Adv_Arr[12] := FALSE;
   S704_LM_DC_2ND_CLAMP6.Visu_Adv_Arr[13] := FALSE;
   S704_LM_DC_2ND_CLAMP6.Visu_Adv_Arr[14] := FALSE;
   S704_LM_DC_2ND_CLAMP6.Visu_Adv_Arr[15] := FALSE;
   S704_LM_DC_2ND_CLAMP6.Visu_Ret_Arr[0] := FALSE;
   S704_LM_DC_2ND_CLAMP6.Visu_Ret_Arr[1] := FALSE;
   S704_LM_DC_2ND_CLAMP6.Visu_Ret_Arr[2] := FALSE;
   S704_LM_DC_2ND_CLAMP6.Visu_Ret_Arr[3] := FALSE;
   S704_LM_DC_2ND_CLAMP6.Visu_Ret_Arr[4] := FALSE;
   S704_LM_DC_2ND_CLAMP6.Visu_Ret_Arr[5] := FALSE;
   S704_LM_DC_2ND_CLAMP6.Visu_Ret_Arr[6] := FALSE;
   S704_LM_DC_2ND_CLAMP6.Visu_Ret_Arr[7] := FALSE;
   S704_LM_DC_2ND_CLAMP6.Visu_Ret_Arr[8] := FALSE;
   S704_LM_DC_2ND_CLAMP6.Visu_Ret_Arr[9] := FALSE;
   S704_LM_DC_2ND_CLAMP6.Visu_Ret_Arr[10] := FALSE;
   S704_LM_DC_2ND_CLAMP6.Visu_Ret_Arr[11] := FALSE;
   S704_LM_DC_2ND_CLAMP6.Visu_Ret_Arr[12] := FALSE;
   S704_LM_DC_2ND_CLAMP6.Visu_Ret_Arr[13] := FALSE;
   S704_LM_DC_2ND_CLAMP6.Visu_Ret_Arr[14] := FALSE;
   S704_LM_DC_2ND_CLAMP6.Visu_Ret_Arr[15] := FALSE;
   S704_LM_DC_2ND_CLAMP6.BLK_Move_Ret := 0;
   S704_LM_DC_2ND_CLAMP6.Enable := FALSE;
   S704_LM_DC_2ND_CLAMP6.Adv_End := FALSE;
   S704_LM_DC_2ND_CLAMP6.Ret_End := FALSE;
   S704_LM_DC_2ND_CLAMP7.Enable_Aux := FALSE;
   S704_LM_DC_2ND_CLAMP7.Adv_Amount := 0;
   S704_LM_DC_2ND_CLAMP7.Ret_Amount := 0;
   S704_LM_DC_2ND_CLAMP7.LS_Adv1 := FALSE;
   S704_LM_DC_2ND_CLAMP7.LS_Ret1 := FALSE;
   S704_LM_DC_2ND_CLAMP7.LS_Adv2 := FALSE;
   S704_LM_DC_2ND_CLAMP7.LS_Ret2 := FALSE;
   S704_LM_DC_2ND_CLAMP7.LS_Adv3 := FALSE;
   S704_LM_DC_2ND_CLAMP7.LS_Ret3 := FALSE;
   S704_LM_DC_2ND_CLAMP7.LS_Adv4 := FALSE;
   S704_LM_DC_2ND_CLAMP7.LS_Ret4 := FALSE;
   S704_LM_DC_2ND_CLAMP7.SOL_Adv := FALSE;
   S704_LM_DC_2ND_CLAMP7.SOL_Ret := FALSE;
   S704_LM_DC_2ND_CLAMP7.M_Ready := FALSE;
   S704_LM_DC_2ND_CLAMP7.T_CHK1 := T#0MS;
   S704_LM_DC_2ND_CLAMP7.T_CHK2 := T#0MS;
   S704_LM_DC_2ND_CLAMP7.PB_Lamp_CHK := FALSE;
   S704_LM_DC_2ND_CLAMP7.PB_Error_Rst := FALSE;
   S704_LM_DC_2ND_CLAMP7.M_FLICK := FALSE;
   S704_LM_DC_2ND_CLAMP7.M_Adv_Err := FALSE;
   S704_LM_DC_2ND_CLAMP7.M_Ret_Err := FALSE;
   S704_LM_DC_2ND_CLAMP7.LP_Adv := FALSE;
   S704_LM_DC_2ND_CLAMP7.LP_Ret := FALSE;
   S704_LM_DC_2ND_CLAMP7.Visu_Adv := W#16#0;
   S704_LM_DC_2ND_CLAMP7.Visu_Ret := W#16#0;
   S704_LM_DC_2ND_CLAMP7.Error_T1.IN := FALSE;
   S704_LM_DC_2ND_CLAMP7.Error_T1.PT := T#0MS;
   S704_LM_DC_2ND_CLAMP7.Error_T1.Q := FALSE;
   S704_LM_DC_2ND_CLAMP7.Error_T1.ET := T#0MS;
   S704_LM_DC_2ND_CLAMP7.Error_T1.STATE := B#16#0;
   S704_LM_DC_2ND_CLAMP7.Error_T1.STIME := T#0MS;
   S704_LM_DC_2ND_CLAMP7.Error_T1.ATIME := T#0MS;
   S704_LM_DC_2ND_CLAMP7.Error_T2.IN := FALSE;
   S704_LM_DC_2ND_CLAMP7.Error_T2.PT := T#0MS;
   S704_LM_DC_2ND_CLAMP7.Error_T2.Q := FALSE;
   S704_LM_DC_2ND_CLAMP7.Error_T2.ET := T#0MS;
   S704_LM_DC_2ND_CLAMP7.Error_T2.STATE := B#16#0;
   S704_LM_DC_2ND_CLAMP7.Error_T2.STIME := T#0MS;
   S704_LM_DC_2ND_CLAMP7.Error_T2.ATIME := T#0MS;
   S704_LM_DC_2ND_CLAMP7.CHK_Aux1 := FALSE;
   S704_LM_DC_2ND_CLAMP7.CHK_Aux2 := FALSE;
   S704_LM_DC_2ND_CLAMP7.Error_T1_DN := FALSE;
   S704_LM_DC_2ND_CLAMP7.Error_T2_DN := FALSE;
   S704_LM_DC_2ND_CLAMP7.Adv_Memo := FALSE;
   S704_LM_DC_2ND_CLAMP7.Visu_Adv_Arr[0] := FALSE;
   S704_LM_DC_2ND_CLAMP7.Visu_Adv_Arr[1] := FALSE;
   S704_LM_DC_2ND_CLAMP7.Visu_Adv_Arr[2] := FALSE;
   S704_LM_DC_2ND_CLAMP7.Visu_Adv_Arr[3] := FALSE;
   S704_LM_DC_2ND_CLAMP7.Visu_Adv_Arr[4] := FALSE;
   S704_LM_DC_2ND_CLAMP7.Visu_Adv_Arr[5] := FALSE;
   S704_LM_DC_2ND_CLAMP7.Visu_Adv_Arr[6] := FALSE;
   S704_LM_DC_2ND_CLAMP7.Visu_Adv_Arr[7] := FALSE;
   S704_LM_DC_2ND_CLAMP7.Visu_Adv_Arr[8] := FALSE;
   S704_LM_DC_2ND_CLAMP7.Visu_Adv_Arr[9] := FALSE;
   S704_LM_DC_2ND_CLAMP7.Visu_Adv_Arr[10] := FALSE;
   S704_LM_DC_2ND_CLAMP7.Visu_Adv_Arr[11] := FALSE;
   S704_LM_DC_2ND_CLAMP7.Visu_Adv_Arr[12] := FALSE;
   S704_LM_DC_2ND_CLAMP7.Visu_Adv_Arr[13] := FALSE;
   S704_LM_DC_2ND_CLAMP7.Visu_Adv_Arr[14] := FALSE;
   S704_LM_DC_2ND_CLAMP7.Visu_Adv_Arr[15] := FALSE;
   S704_LM_DC_2ND_CLAMP7.Visu_Ret_Arr[0] := FALSE;
   S704_LM_DC_2ND_CLAMP7.Visu_Ret_Arr[1] := FALSE;
   S704_LM_DC_2ND_CLAMP7.Visu_Ret_Arr[2] := FALSE;
   S704_LM_DC_2ND_CLAMP7.Visu_Ret_Arr[3] := FALSE;
   S704_LM_DC_2ND_CLAMP7.Visu_Ret_Arr[4] := FALSE;
   S704_LM_DC_2ND_CLAMP7.Visu_Ret_Arr[5] := FALSE;
   S704_LM_DC_2ND_CLAMP7.Visu_Ret_Arr[6] := FALSE;
   S704_LM_DC_2ND_CLAMP7.Visu_Ret_Arr[7] := FALSE;
   S704_LM_DC_2ND_CLAMP7.Visu_Ret_Arr[8] := FALSE;
   S704_LM_DC_2ND_CLAMP7.Visu_Ret_Arr[9] := FALSE;
   S704_LM_DC_2ND_CLAMP7.Visu_Ret_Arr[10] := FALSE;
   S704_LM_DC_2ND_CLAMP7.Visu_Ret_Arr[11] := FALSE;
   S704_LM_DC_2ND_CLAMP7.Visu_Ret_Arr[12] := FALSE;
   S704_LM_DC_2ND_CLAMP7.Visu_Ret_Arr[13] := FALSE;
   S704_LM_DC_2ND_CLAMP7.Visu_Ret_Arr[14] := FALSE;
   S704_LM_DC_2ND_CLAMP7.Visu_Ret_Arr[15] := FALSE;
   S704_LM_DC_2ND_CLAMP7.BLK_Move_Ret := 0;
   S704_LM_DC_2ND_CLAMP7.Enable := FALSE;
   S704_LM_DC_2ND_CLAMP7.Adv_End := FALSE;
   S704_LM_DC_2ND_CLAMP7.Ret_End := FALSE;
   S704_LM_DC_1ST_CLAMP5.Enable_Aux := FALSE;
   S704_LM_DC_1ST_CLAMP5.Adv_Amount := 0;
   S704_LM_DC_1ST_CLAMP5.Ret_Amount := 0;
   S704_LM_DC_1ST_CLAMP5.LS_Adv1 := FALSE;
   S704_LM_DC_1ST_CLAMP5.LS_Ret1 := FALSE;
   S704_LM_DC_1ST_CLAMP5.LS_Adv2 := FALSE;
   S704_LM_DC_1ST_CLAMP5.LS_Ret2 := FALSE;
   S704_LM_DC_1ST_CLAMP5.LS_Adv3 := FALSE;
   S704_LM_DC_1ST_CLAMP5.LS_Ret3 := FALSE;
   S704_LM_DC_1ST_CLAMP5.LS_Adv4 := FALSE;
   S704_LM_DC_1ST_CLAMP5.LS_Ret4 := FALSE;
   S704_LM_DC_1ST_CLAMP5.SOL_Adv := FALSE;
   S704_LM_DC_1ST_CLAMP5.SOL_Ret := FALSE;
   S704_LM_DC_1ST_CLAMP5.M_Ready := FALSE;
   S704_LM_DC_1ST_CLAMP5.T_CHK1 := T#0MS;
   S704_LM_DC_1ST_CLAMP5.T_CHK2 := T#0MS;
   S704_LM_DC_1ST_CLAMP5.PB_Lamp_CHK := FALSE;
   S704_LM_DC_1ST_CLAMP5.PB_Error_Rst := FALSE;
   S704_LM_DC_1ST_CLAMP5.M_FLICK := FALSE;
   S704_LM_DC_1ST_CLAMP5.M_Adv_Err := FALSE;
   S704_LM_DC_1ST_CLAMP5.M_Ret_Err := FALSE;
   S704_LM_DC_1ST_CLAMP5.LP_Adv := FALSE;
   S704_LM_DC_1ST_CLAMP5.LP_Ret := FALSE;
   S704_LM_DC_1ST_CLAMP5.Visu_Adv := W#16#0;
   S704_LM_DC_1ST_CLAMP5.Visu_Ret := W#16#0;
   S704_LM_DC_1ST_CLAMP5.Error_T1.IN := FALSE;
   S704_LM_DC_1ST_CLAMP5.Error_T1.PT := T#0MS;
   S704_LM_DC_1ST_CLAMP5.Error_T1.Q := FALSE;
   S704_LM_DC_1ST_CLAMP5.Error_T1.ET := T#0MS;
   S704_LM_DC_1ST_CLAMP5.Error_T1.STATE := B#16#0;
   S704_LM_DC_1ST_CLAMP5.Error_T1.STIME := T#0MS;
   S704_LM_DC_1ST_CLAMP5.Error_T1.ATIME := T#0MS;
   S704_LM_DC_1ST_CLAMP5.Error_T2.IN := FALSE;
   S704_LM_DC_1ST_CLAMP5.Error_T2.PT := T#0MS;
   S704_LM_DC_1ST_CLAMP5.Error_T2.Q := FALSE;
   S704_LM_DC_1ST_CLAMP5.Error_T2.ET := T#0MS;
   S704_LM_DC_1ST_CLAMP5.Error_T2.STATE := B#16#0;
   S704_LM_DC_1ST_CLAMP5.Error_T2.STIME := T#0MS;
   S704_LM_DC_1ST_CLAMP5.Error_T2.ATIME := T#0MS;
   S704_LM_DC_1ST_CLAMP5.CHK_Aux1 := FALSE;
   S704_LM_DC_1ST_CLAMP5.CHK_Aux2 := FALSE;
   S704_LM_DC_1ST_CLAMP5.Error_T1_DN := FALSE;
   S704_LM_DC_1ST_CLAMP5.Error_T2_DN := FALSE;
   S704_LM_DC_1ST_CLAMP5.Adv_Memo := FALSE;
   S704_LM_DC_1ST_CLAMP5.Visu_Adv_Arr[0] := FALSE;
   S704_LM_DC_1ST_CLAMP5.Visu_Adv_Arr[1] := FALSE;
   S704_LM_DC_1ST_CLAMP5.Visu_Adv_Arr[2] := FALSE;
   S704_LM_DC_1ST_CLAMP5.Visu_Adv_Arr[3] := FALSE;
   S704_LM_DC_1ST_CLAMP5.Visu_Adv_Arr[4] := FALSE;
   S704_LM_DC_1ST_CLAMP5.Visu_Adv_Arr[5] := FALSE;
   S704_LM_DC_1ST_CLAMP5.Visu_Adv_Arr[6] := FALSE;
   S704_LM_DC_1ST_CLAMP5.Visu_Adv_Arr[7] := FALSE;
   S704_LM_DC_1ST_CLAMP5.Visu_Adv_Arr[8] := FALSE;
   S704_LM_DC_1ST_CLAMP5.Visu_Adv_Arr[9] := FALSE;
   S704_LM_DC_1ST_CLAMP5.Visu_Adv_Arr[10] := FALSE;
   S704_LM_DC_1ST_CLAMP5.Visu_Adv_Arr[11] := FALSE;
   S704_LM_DC_1ST_CLAMP5.Visu_Adv_Arr[12] := FALSE;
   S704_LM_DC_1ST_CLAMP5.Visu_Adv_Arr[13] := FALSE;
   S704_LM_DC_1ST_CLAMP5.Visu_Adv_Arr[14] := FALSE;
   S704_LM_DC_1ST_CLAMP5.Visu_Adv_Arr[15] := FALSE;
   S704_LM_DC_1ST_CLAMP5.Visu_Ret_Arr[0] := FALSE;
   S704_LM_DC_1ST_CLAMP5.Visu_Ret_Arr[1] := FALSE;
   S704_LM_DC_1ST_CLAMP5.Visu_Ret_Arr[2] := FALSE;
   S704_LM_DC_1ST_CLAMP5.Visu_Ret_Arr[3] := FALSE;
   S704_LM_DC_1ST_CLAMP5.Visu_Ret_Arr[4] := FALSE;
   S704_LM_DC_1ST_CLAMP5.Visu_Ret_Arr[5] := FALSE;
   S704_LM_DC_1ST_CLAMP5.Visu_Ret_Arr[6] := FALSE;
   S704_LM_DC_1ST_CLAMP5.Visu_Ret_Arr[7] := FALSE;
   S704_LM_DC_1ST_CLAMP5.Visu_Ret_Arr[8] := FALSE;
   S704_LM_DC_1ST_CLAMP5.Visu_Ret_Arr[9] := FALSE;
   S704_LM_DC_1ST_CLAMP5.Visu_Ret_Arr[10] := FALSE;
   S704_LM_DC_1ST_CLAMP5.Visu_Ret_Arr[11] := FALSE;
   S704_LM_DC_1ST_CLAMP5.Visu_Ret_Arr[12] := FALSE;
   S704_LM_DC_1ST_CLAMP5.Visu_Ret_Arr[13] := FALSE;
   S704_LM_DC_1ST_CLAMP5.Visu_Ret_Arr[14] := FALSE;
   S704_LM_DC_1ST_CLAMP5.Visu_Ret_Arr[15] := FALSE;
   S704_LM_DC_1ST_CLAMP5.BLK_Move_Ret := 0;
   S704_LM_DC_1ST_CLAMP5.Enable := FALSE;
   S704_LM_DC_1ST_CLAMP5.Adv_End := FALSE;
   S704_LM_DC_1ST_CLAMP5.Ret_End := FALSE;
END_DATA_BLOCK

FUNCTION FC 143 : VOID
TITLE =
VERSION : 0.1

BEGIN
NETWORK
TITLE =
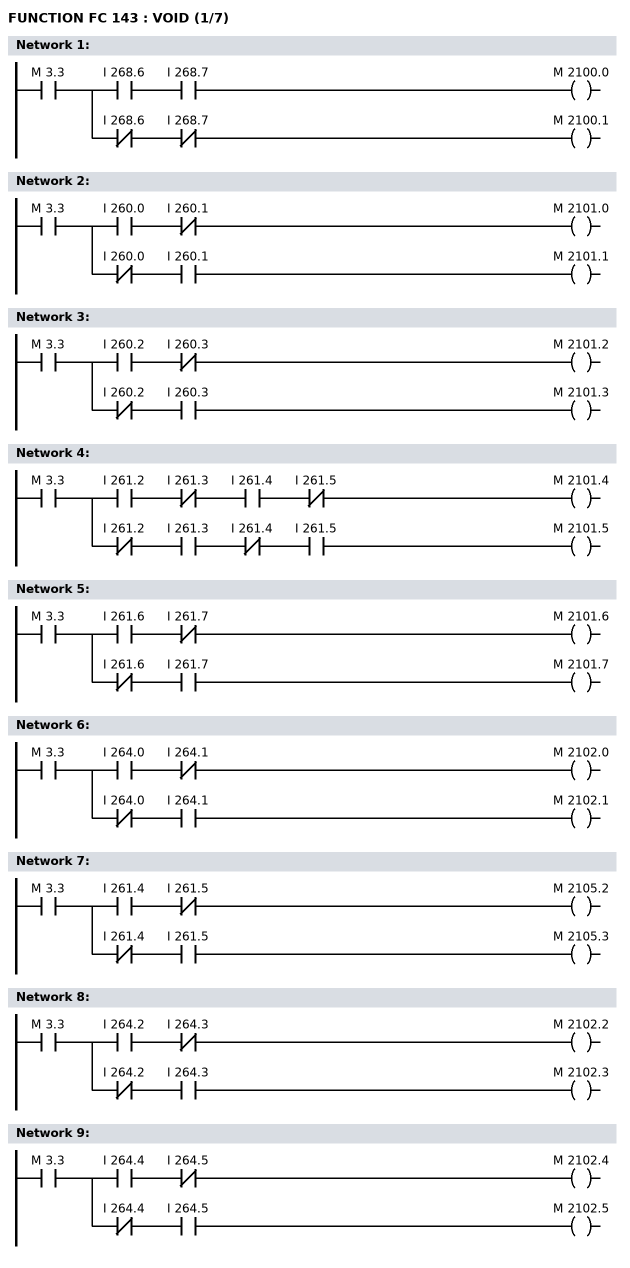

      A     M      3.3;
      =     L      0.0;
      A     L      0.0;
      A     I    268.6;
      A     I    268.7;
      =     M   2100.0;
      A     L      0.0;
      AN    I    268.6;
      AN    I    268.7;
      =     M   2100.1;
NETWORK
TITLE =

      A     M      3.3;
      =     L      0.0;
      A     L      0.0;
      A     I    260.0;
      AN    I    260.1;
      =     M   2101.0;
      A     L      0.0;
      AN    I    260.0;
      A     I    260.1;
      =     M   2101.1;
NETWORK
TITLE =

      A     M      3.3;
      =     L      0.0;
      A     L      0.0;
      A     I    260.2;
      AN    I    260.3;
      =     M   2101.2;
      A     L      0.0;
      AN    I    260.2;
      A     I    260.3;
      =     M   2101.3;
NETWORK
TITLE =

      A     M      3.3;
      =     L      0.0;
      A     L      0.0;
      A     I    261.2;
      AN    I    261.3;
      A     I    261.4;
      AN    I    261.5;
      =     M   2101.4;
      A     L      0.0;
      AN    I    261.2;
      A     I    261.3;
      AN    I    261.4;
      A     I    261.5;
      =     M   2101.5;
NETWORK
TITLE =

      A     M      3.3;
      =     L      0.0;
      A     L      0.0;
      A     I    261.6;
      AN    I    261.7;
      =     M   2101.6;
      A     L      0.0;
      AN    I    261.6;
      A     I    261.7;
      =     M   2101.7;
NETWORK
TITLE =

      A     M      3.3;
      =     L      0.0;
      A     L      0.0;
      A     I    264.0;
      AN    I    264.1;
      =     M   2102.0;
      A     L      0.0;
      AN    I    264.0;
      A     I    264.1;
      =     M   2102.1;
NETWORK
TITLE =

      A     M      3.3;
      =     L      0.0;
      A     L      0.0;
      A     I    261.4;
      AN    I    261.5;
      =     M   2105.2;
      A     L      0.0;
      AN    I    261.4;
      A     I    261.5;
      =     M   2105.3;
NETWORK
TITLE =

      A     M      3.3;
      =     L      0.0;
      A     L      0.0;
      A     I    264.2;
      AN    I    264.3;
      =     M   2102.2;
      A     L      0.0;
      AN    I    264.2;
      A     I    264.3;
      =     M   2102.3;
NETWORK
TITLE =

      A     M      3.3;
      =     L      0.0;
      A     L      0.0;
      A     I    264.4;
      AN    I    264.5;
      =     M   2102.4;
      A     L      0.0;
      AN    I    264.4;
      A     I    264.5;
      =     M   2102.5;
NETWORK
TITLE =
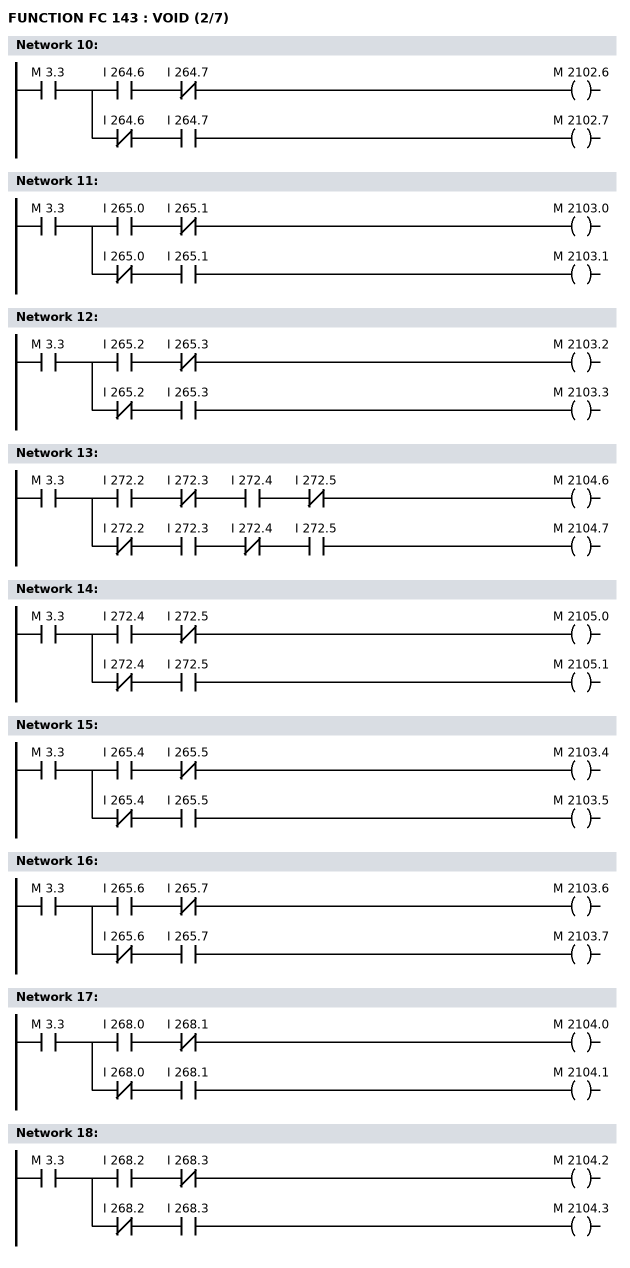

      A     M      3.3;
      =     L      0.0;
      A     L      0.0;
      A     I    264.6;
      AN    I    264.7;
      =     M   2102.6;
      A     L      0.0;
      AN    I    264.6;
      A     I    264.7;
      =     M   2102.7;
NETWORK
TITLE =

      A     M      3.3;
      =     L      0.0;
      A     L      0.0;
      A     I    265.0;
      AN    I    265.1;
      =     M   2103.0;
      A     L      0.0;
      AN    I    265.0;
      A     I    265.1;
      =     M   2103.1;
NETWORK
TITLE =

      A     M      3.3;
      =     L      0.0;
      A     L      0.0;
      A     I    265.2;
      AN    I    265.3;
      =     M   2103.2;
      A     L      0.0;
      AN    I    265.2;
      A     I    265.3;
      =     M   2103.3;
NETWORK
TITLE =

      A     M      3.3;
      =     L      0.0;
      A     L      0.0;
      A     I    272.2;
      AN    I    272.3;
      A     I    272.4;
      AN    I    272.5;
      =     M   2104.6;
      A     L      0.0;
      AN    I    272.2;
      A     I    272.3;
      AN    I    272.4;
      A     I    272.5;
      =     M   2104.7;
NETWORK
TITLE =

      A     M      3.3;
      =     L      0.0;
      A     L      0.0;
      A     I    272.4;
      AN    I    272.5;
      =     M   2105.0;
      A     L      0.0;
      AN    I    272.4;
      A     I    272.5;
      =     M   2105.1;
NETWORK
TITLE =

      A     M      3.3;
      =     L      0.0;
      A     L      0.0;
      A     I    265.4;
      AN    I    265.5;
      =     M   2103.4;
      A     L      0.0;
      AN    I    265.4;
      A     I    265.5;
      =     M   2103.5;
NETWORK
TITLE =

      A     M      3.3;
      =     L      0.0;
      A     L      0.0;
      A     I    265.6;
      AN    I    265.7;
      =     M   2103.6;
      A     L      0.0;
      AN    I    265.6;
      A     I    265.7;
      =     M   2103.7;
NETWORK
TITLE =

      A     M      3.3;
      =     L      0.0;
      A     L      0.0;
      A     I    268.0;
      AN    I    268.1;
      =     M   2104.0;
      A     L      0.0;
      AN    I    268.0;
      A     I    268.1;
      =     M   2104.1;
NETWORK
TITLE =

      A     M      3.3;
      =     L      0.0;
      A     L      0.0;
      A     I    268.2;
      AN    I    268.3;
      =     M   2104.2;
      A     L      0.0;
      AN    I    268.2;
      A     I    268.3;
      =     M   2104.3;
NETWORK
TITLE =
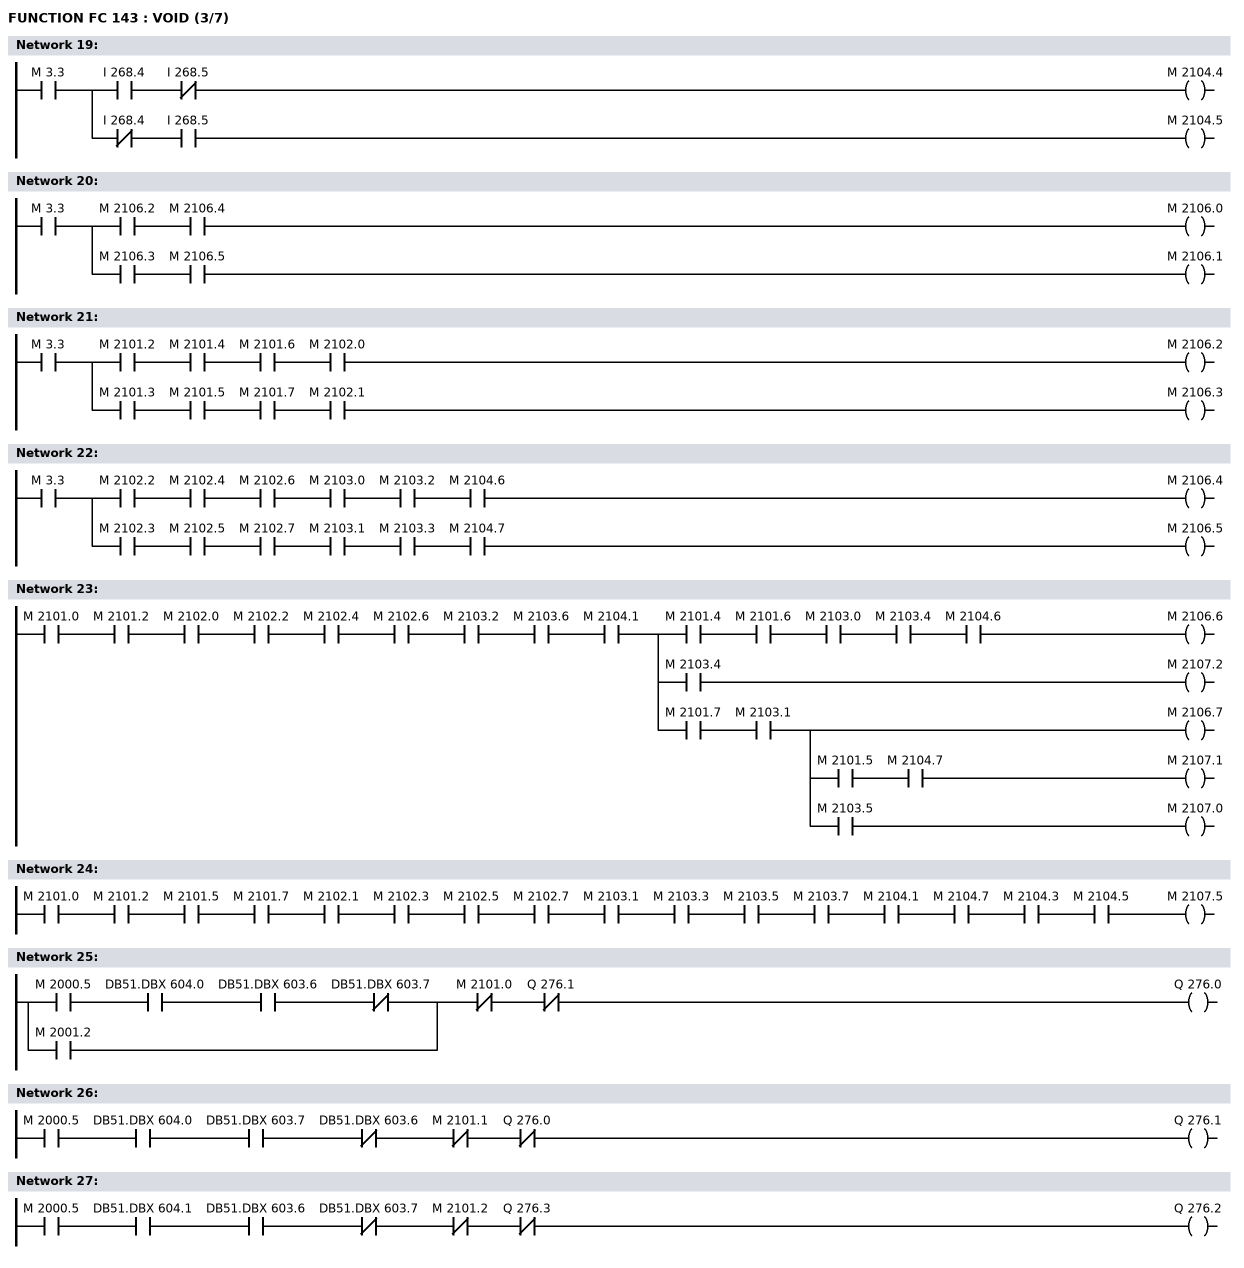

      A     M      3.3;
      =     L      0.0;
      A     L      0.0;
      A     I    268.4;
      AN    I    268.5;
      =     M   2104.4;
      A     L      0.0;
      AN    I    268.4;
      A     I    268.5;
      =     M   2104.5;
NETWORK
TITLE =

      A     M      3.3;
      =     L      0.0;
      A     L      0.0;
      A     M   2106.2;
      A     M   2106.4;
      =     M   2106.0;
      A     L      0.0;
      A     M   2106.3;
      A     M   2106.5;
      =     M   2106.1;
NETWORK
TITLE =

      A     M      3.3;
      =     L      0.0;
      A     L      0.0;
      A     M   2101.2;
      A     M   2101.4;
      A     M   2101.6;
      A     M   2102.0;
      =     M   2106.2;
      A     L      0.0;
      A     M   2101.3;
      A     M   2101.5;
      A     M   2101.7;
      A     M   2102.1;
      =     M   2106.3;
NETWORK
TITLE =

      A     M      3.3;
      =     L      0.0;
      A     L      0.0;
      A     M   2102.2;
      A     M   2102.4;
      A     M   2102.6;
      A     M   2103.0;
      A     M   2103.2;
      A     M   2104.6;
      =     M   2106.4;
      A     L      0.0;
      A     M   2102.3;
      A     M   2102.5;
      A     M   2102.7;
      A     M   2103.1;
      A     M   2103.3;
      A     M   2104.7;
      =     M   2106.5;
NETWORK
TITLE =

      A     M   2101.0;
      A     M   2101.2;
      A     M   2102.0;
      A     M   2102.2;
      A     M   2102.4;
      A     M   2102.6;
      A     M   2103.2;
      A     M   2103.6;
      A     M   2104.1;
      =     L      0.0;
      A     L      0.0;
      A     M   2101.4;
      A     M   2101.6;
      A     M   2103.0;
      A     M   2103.4;
      A     M   2104.6;
      =     M   2106.6;
      A     L      0.0;
      A     M   2103.4;
      =     M   2107.2;
      A     L      0.0;
      A     M   2101.7;
      A     M   2103.1;
      =     L      0.1;
      A     L      0.1;
      BLD   102;
      =     M   2106.7;
      A     L      0.1;
      A     M   2101.5;
      A     M   2104.7;
      =     M   2107.1;
      A     L      0.1;
      A     M   2103.5;
      =     M   2107.0;
NETWORK
TITLE =

      A     M   2101.0;
      A     M   2101.2;
      A     M   2101.5;
      A     M   2101.7;
      A     M   2102.1;
      A     M   2102.3;
      A     M   2102.5;
      A     M   2102.7;
      A     M   2103.1;
      A     M   2103.3;
      A     M   2103.5;
      A     M   2103.7;
      A     M   2104.1;
      A     M   2104.7;
      A     M   2104.3;
      A     M   2104.5;
      =     M   2107.5;
NETWORK
TITLE =

      A(    ;
      A     M   2000.5;
      A     DB51.DBX  604.0;
      A     DB51.DBX  603.6;
      AN    DB51.DBX  603.7;
      O     M   2001.2;
      )     ;
      AN    M   2101.0;
      AN    Q    276.1;
      =     Q    276.0;
NETWORK
TITLE =

      A     M   2000.5;
      A     DB51.DBX  604.0;
      A     DB51.DBX  603.7;
      AN    DB51.DBX  603.6;
      AN    M   2101.1;
      AN    Q    276.0;
      =     Q    276.1;
NETWORK
TITLE =

      A     M   2000.5;
      A     DB51.DBX  604.1;
      A     DB51.DBX  603.6;
      AN    DB51.DBX  603.7;
      AN    M   2101.2;
      AN    Q    276.3;
      =     Q    276.2;
NETWORK
TITLE =
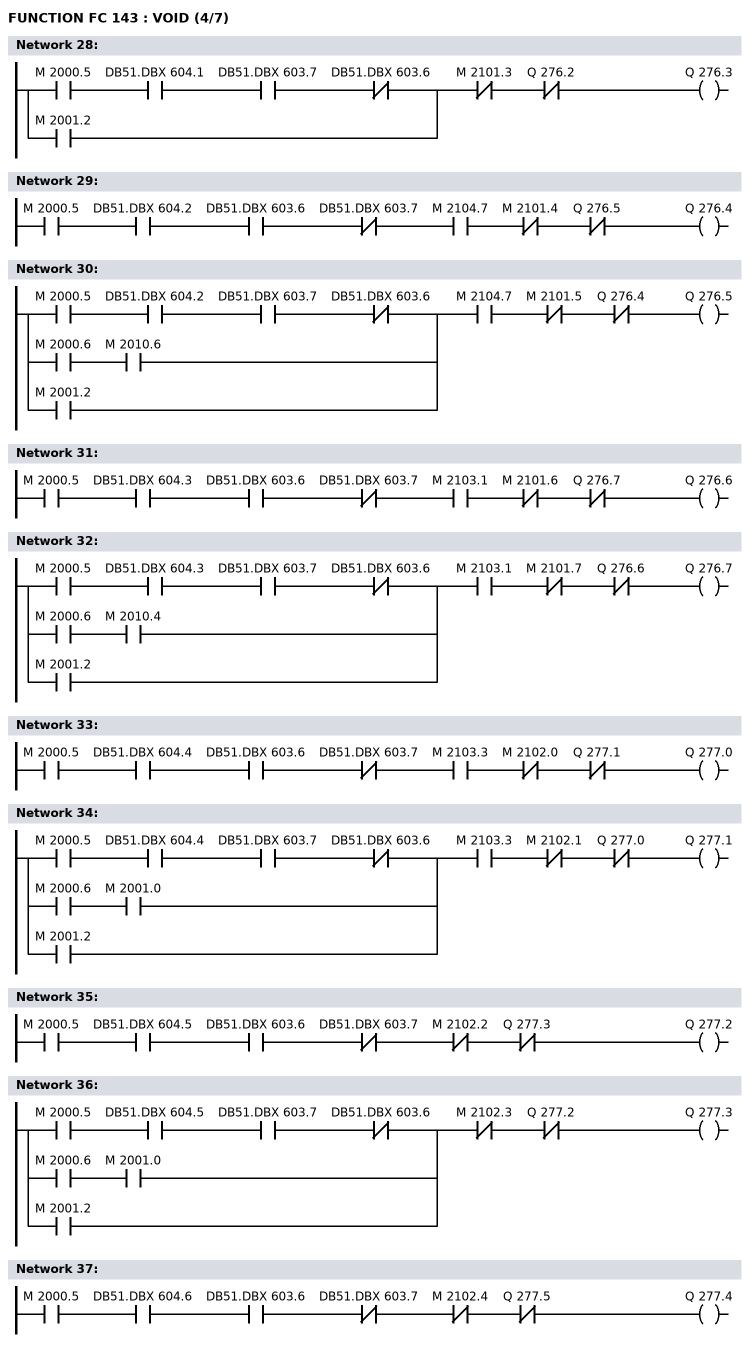

      A(    ;
      A     M   2000.5;
      A     DB51.DBX  604.1;
      A     DB51.DBX  603.7;
      AN    DB51.DBX  603.6;
      O     M   2001.2;
      )     ;
      AN    M   2101.3;
      AN    Q    276.2;
      =     Q    276.3;
NETWORK
TITLE =

      A     M   2000.5;
      A     DB51.DBX  604.2;
      A     DB51.DBX  603.6;
      AN    DB51.DBX  603.7;
      A     M   2104.7;
      AN    M   2101.4;
      AN    Q    276.5;
      =     Q    276.4;
NETWORK
TITLE =

      A(    ;
      A     M   2000.5;
      A     DB51.DBX  604.2;
      A     DB51.DBX  603.7;
      AN    DB51.DBX  603.6;
      O     ;
      A     M   2000.6;
      A     M   2010.6;
      O     M   2001.2;
      )     ;
      A     M   2104.7;
      AN    M   2101.5;
      AN    Q    276.4;
      =     Q    276.5;
NETWORK
TITLE =

      A     M   2000.5;
      A     DB51.DBX  604.3;
      A     DB51.DBX  603.6;
      AN    DB51.DBX  603.7;
      A     M   2103.1;
      AN    M   2101.6;
      AN    Q    276.7;
      =     Q    276.6;
NETWORK
TITLE =

      A(    ;
      A     M   2000.5;
      A     DB51.DBX  604.3;
      A     DB51.DBX  603.7;
      AN    DB51.DBX  603.6;
      O     ;
      A     M   2000.6;
      A     M   2010.4;
      O     M   2001.2;
      )     ;
      A     M   2103.1;
      AN    M   2101.7;
      AN    Q    276.6;
      =     Q    276.7;
NETWORK
TITLE =

      A     M   2000.5;
      A     DB51.DBX  604.4;
      A     DB51.DBX  603.6;
      AN    DB51.DBX  603.7;
      A     M   2103.3;
      AN    M   2102.0;
      AN    Q    277.1;
      =     Q    277.0;
NETWORK
TITLE =

      A(    ;
      A     M   2000.5;
      A     DB51.DBX  604.4;
      A     DB51.DBX  603.7;
      AN    DB51.DBX  603.6;
      O     ;
      A     M   2000.6;
      A     M   2001.0;
      O     M   2001.2;
      )     ;
      A     M   2103.3;
      AN    M   2102.1;
      AN    Q    277.0;
      =     Q    277.1;
NETWORK
TITLE =

      A     M   2000.5;
      A     DB51.DBX  604.5;
      A     DB51.DBX  603.6;
      AN    DB51.DBX  603.7;
      AN    M   2102.2;
      AN    Q    277.3;
      =     Q    277.2;
NETWORK
TITLE =

      A(    ;
      A     M   2000.5;
      A     DB51.DBX  604.5;
      A     DB51.DBX  603.7;
      AN    DB51.DBX  603.6;
      O     ;
      A     M   2000.6;
      A     M   2001.0;
      O     M   2001.2;
      )     ;
      AN    M   2102.3;
      AN    Q    277.2;
      =     Q    277.3;
NETWORK
TITLE =

      A     M   2000.5;
      A     DB51.DBX  604.6;
      A     DB51.DBX  603.6;
      AN    DB51.DBX  603.7;
      AN    M   2102.4;
      AN    Q    277.5;
      =     Q    277.4;
NETWORK
TITLE =
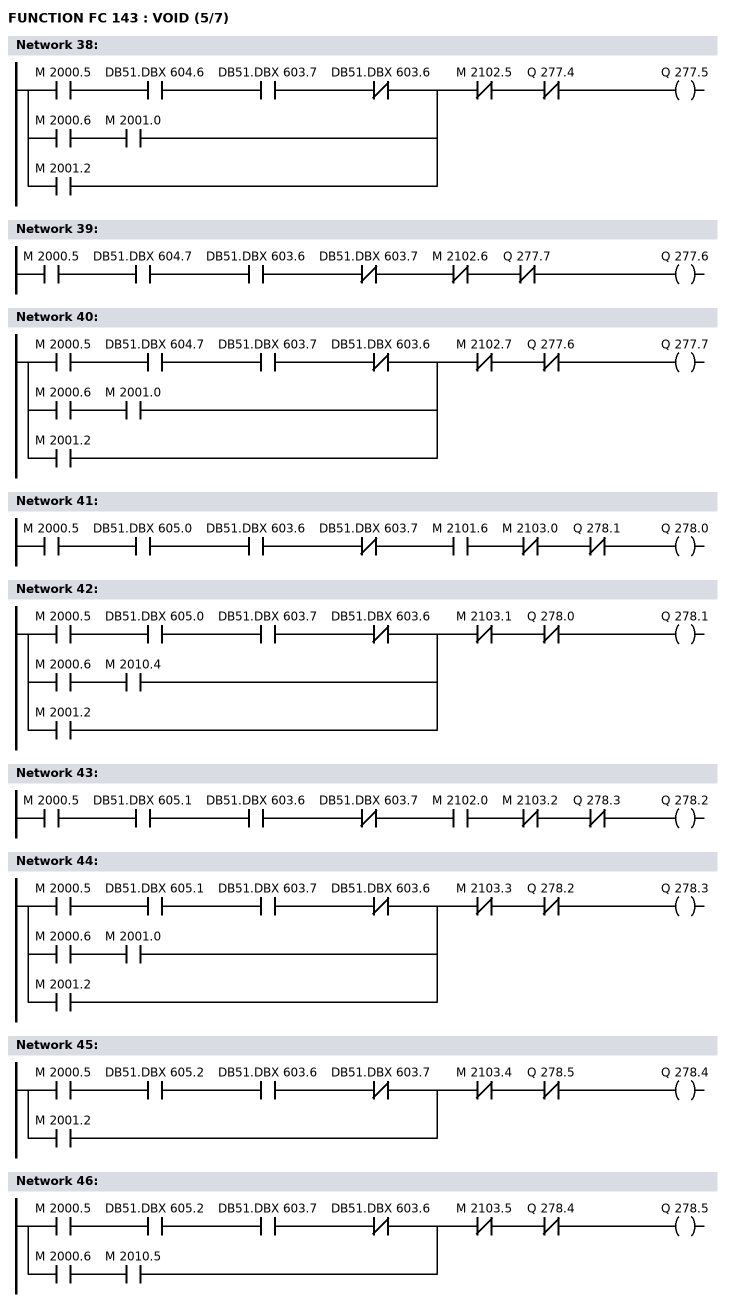

      A(    ;
      A     M   2000.5;
      A     DB51.DBX  604.6;
      A     DB51.DBX  603.7;
      AN    DB51.DBX  603.6;
      O     ;
      A     M   2000.6;
      A     M   2001.0;
      O     M   2001.2;
      )     ;
      AN    M   2102.5;
      AN    Q    277.4;
      =     Q    277.5;
NETWORK
TITLE =

      A     M   2000.5;
      A     DB51.DBX  604.7;
      A     DB51.DBX  603.6;
      AN    DB51.DBX  603.7;
      AN    M   2102.6;
      AN    Q    277.7;
      =     Q    277.6;
NETWORK
TITLE =

      A(    ;
      A     M   2000.5;
      A     DB51.DBX  604.7;
      A     DB51.DBX  603.7;
      AN    DB51.DBX  603.6;
      O     ;
      A     M   2000.6;
      A     M   2001.0;
      O     M   2001.2;
      )     ;
      AN    M   2102.7;
      AN    Q    277.6;
      =     Q    277.7;
NETWORK
TITLE =

      A     M   2000.5;
      A     DB51.DBX  605.0;
      A     DB51.DBX  603.6;
      AN    DB51.DBX  603.7;
      A     M   2101.6;
      AN    M   2103.0;
      AN    Q    278.1;
      =     Q    278.0;
NETWORK
TITLE =

      A(    ;
      A     M   2000.5;
      A     DB51.DBX  605.0;
      A     DB51.DBX  603.7;
      AN    DB51.DBX  603.6;
      O     ;
      A     M   2000.6;
      A     M   2010.4;
      O     M   2001.2;
      )     ;
      AN    M   2103.1;
      AN    Q    278.0;
      =     Q    278.1;
NETWORK
TITLE =

      A     M   2000.5;
      A     DB51.DBX  605.1;
      A     DB51.DBX  603.6;
      AN    DB51.DBX  603.7;
      A     M   2102.0;
      AN    M   2103.2;
      AN    Q    278.3;
      =     Q    278.2;
NETWORK
TITLE =

      A(    ;
      A     M   2000.5;
      A     DB51.DBX  605.1;
      A     DB51.DBX  603.7;
      AN    DB51.DBX  603.6;
      O     ;
      A     M   2000.6;
      A     M   2001.0;
      O     M   2001.2;
      )     ;
      AN    M   2103.3;
      AN    Q    278.2;
      =     Q    278.3;
NETWORK
TITLE =

      A(    ;
      A     M   2000.5;
      A     DB51.DBX  605.2;
      A     DB51.DBX  603.6;
      AN    DB51.DBX  603.7;
      O     M   2001.2;
      )     ;
      AN    M   2103.4;
      AN    Q    278.5;
      =     Q    278.4;
NETWORK
TITLE =

      A(    ;
      A     M   2000.5;
      A     DB51.DBX  605.2;
      A     DB51.DBX  603.7;
      AN    DB51.DBX  603.6;
      O     ;
      A     M   2000.6;
      A     M   2010.5;
      )     ;
      AN    M   2103.5;
      AN    Q    278.4;
      =     Q    278.5;
NETWORK
TITLE =
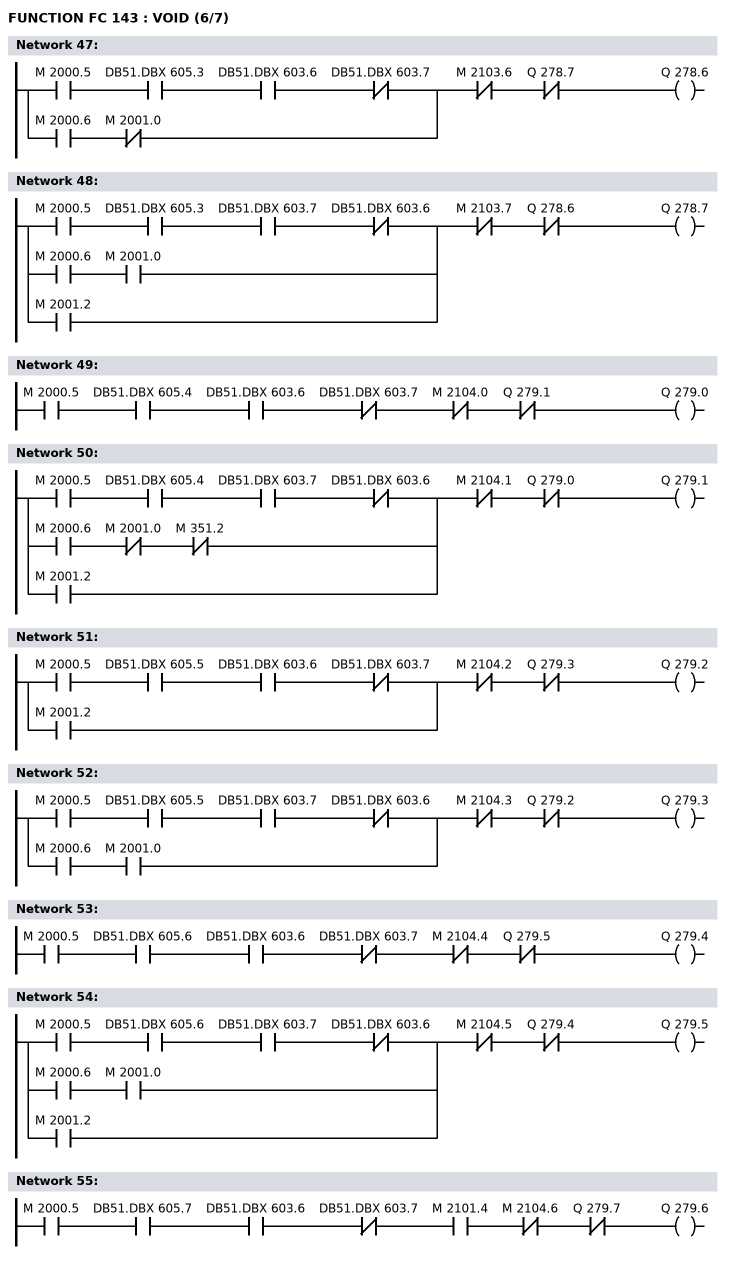

      A(    ;
      A     M   2000.5;
      A     DB51.DBX  605.3;
      A     DB51.DBX  603.6;
      AN    DB51.DBX  603.7;
      O     ;
      A     M   2000.6;
      AN    M   2001.0;
      )     ;
      AN    M   2103.6;
      AN    Q    278.7;
      =     Q    278.6;
NETWORK
TITLE =

      A(    ;
      A     M   2000.5;
      A     DB51.DBX  605.3;
      A     DB51.DBX  603.7;
      AN    DB51.DBX  603.6;
      O     ;
      A     M   2000.6;
      A     M   2001.0;
      O     M   2001.2;
      )     ;
      AN    M   2103.7;
      AN    Q    278.6;
      =     Q    278.7;
NETWORK
TITLE =

      A     M   2000.5;
      A     DB51.DBX  605.4;
      A     DB51.DBX  603.6;
      AN    DB51.DBX  603.7;
      AN    M   2104.0;
      AN    Q    279.1;
      =     Q    279.0;
NETWORK
TITLE =

      A(    ;
      A     M   2000.5;
      A     DB51.DBX  605.4;
      A     DB51.DBX  603.7;
      AN    DB51.DBX  603.6;
      O     ;
      A     M   2000.6;
      AN    M   2001.0;
      AN    M    351.2;
      O     M   2001.2;
      )     ;
      AN    M   2104.1;
      AN    Q    279.0;
      =     Q    279.1;
NETWORK
TITLE =

      A(    ;
      A     M   2000.5;
      A     DB51.DBX  605.5;
      A     DB51.DBX  603.6;
      AN    DB51.DBX  603.7;
      O     M   2001.2;
      )     ;
      AN    M   2104.2;
      AN    Q    279.3;
      =     Q    279.2;
NETWORK
TITLE =

      A(    ;
      A     M   2000.5;
      A     DB51.DBX  605.5;
      A     DB51.DBX  603.7;
      AN    DB51.DBX  603.6;
      O     ;
      A     M   2000.6;
      A     M   2001.0;
      )     ;
      AN    M   2104.3;
      AN    Q    279.2;
      =     Q    279.3;
NETWORK
TITLE =

      A     M   2000.5;
      A     DB51.DBX  605.6;
      A     DB51.DBX  603.6;
      AN    DB51.DBX  603.7;
      AN    M   2104.4;
      AN    Q    279.5;
      =     Q    279.4;
NETWORK
TITLE =

      A(    ;
      A     M   2000.5;
      A     DB51.DBX  605.6;
      A     DB51.DBX  603.7;
      AN    DB51.DBX  603.6;
      O     ;
      A     M   2000.6;
      A     M   2001.0;
      O     M   2001.2;
      )     ;
      AN    M   2104.5;
      AN    Q    279.4;
      =     Q    279.5;
NETWORK
TITLE =

      A     M   2000.5;
      A     DB51.DBX  605.7;
      A     DB51.DBX  603.6;
      AN    DB51.DBX  603.7;
      A     M   2101.4;
      AN    M   2104.6;
      AN    Q    279.7;
      =     Q    279.6;
NETWORK
TITLE =
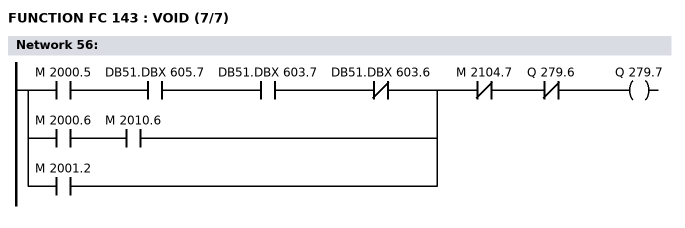

      A(    ;
      A     M   2000.5;
      A     DB51.DBX  605.7;
      A     DB51.DBX  603.7;
      AN    DB51.DBX  603.6;
      O     ;
      A     M   2000.6;
      A     M   2010.6;
      O     M   2001.2;
      )     ;
      AN    M   2104.7;
      AN    Q    279.6;
      =     Q    279.7;
END_FUNCTION

FUNCTION_BLOCK FB 144
TITLE =
VERSION : 0.1


VAR
  S704_TL_DC_PIN : FB 426;
  S704_TL_DC_LATCH1 : FB 426;
  S704_TL_DC_LATCH2 : FB 426;
  S704_TL_DC_1ST_CLAMP1 : FB 426;
  S704_TL_DC_1ST_CLAMP2 : FB 426;
  S704_TL_DC_1ST_CLAMP3 : FB 426;
  S704_TL_DC_2ND_CLAMP1 : FB 426;
  S704_TL_DC_2ND_CLAMP2 : FB 426;
  S704_TL_DC_U261 : FB 426;
  S704_TL_DC_U261_CLAMP : FB 426;
  S704_TL_DC_U269 : FB 426;
  S704_TL_DC_U269_CLAMP : FB 426;
  S704_TL_DC_3RD_CLAMP : FB 426;
  S704_TL_DC_U262_1_UP_DN : FB 426;
  S704_TL_DC_U262_1 : FB 426;
  S704_TL_DC_U262_1_CLAMP : FB 426;
  S704_TL_DC_U261_2_CLAMP : FB 426;
END_VAR
BEGIN
NETWORK
TITLE =
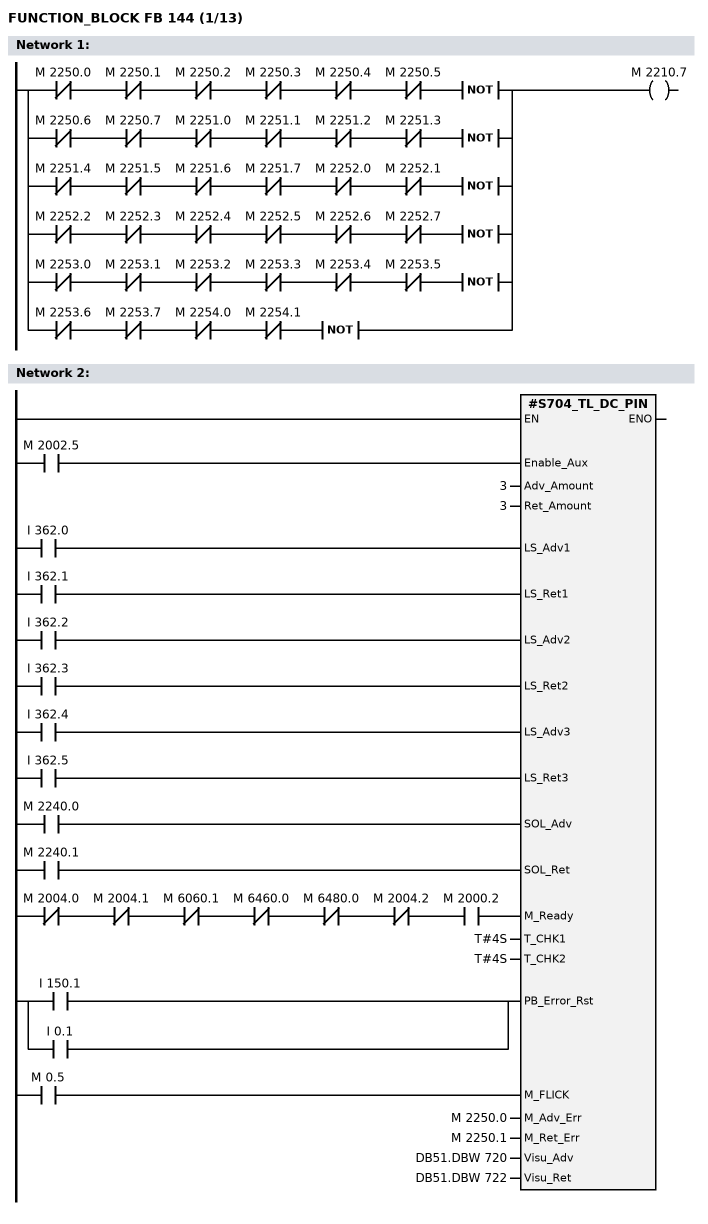

      AN    M   2250.0;
      AN    M   2250.1;
      AN    M   2250.2;
      AN    M   2250.3;
      AN    M   2250.4;
      AN    M   2250.5;
      NOT   ;
      O(    ;
      AN    M   2250.6;
      AN    M   2250.7;
      AN    M   2251.0;
      AN    M   2251.1;
      AN    M   2251.2;
      AN    M   2251.3;
      NOT   ;
      )     ;
      O(    ;
      AN    M   2251.4;
      AN    M   2251.5;
      AN    M   2251.6;
      AN    M   2251.7;
      AN    M   2252.0;
      AN    M   2252.1;
      NOT   ;
      )     ;
      O(    ;
      AN    M   2252.2;
      AN    M   2252.3;
      AN    M   2252.4;
      AN    M   2252.5;
      AN    M   2252.6;
      AN    M   2252.7;
      NOT   ;
      )     ;
      O(    ;
      AN    M   2253.0;
      AN    M   2253.1;
      AN    M   2253.2;
      AN    M   2253.3;
      AN    M   2253.4;
      AN    M   2253.5;
      NOT   ;
      )     ;
      O(    ;
      AN    M   2253.6;
      AN    M   2253.7;
      AN    M   2254.0;
      AN    M   2254.1;
      NOT   ;
      )     ;
      =     M   2210.7;
NETWORK
TITLE =

      A     M   2002.5;
      =     L      0.0;
      BLD   103;
      A     I    362.0;
      =     L      0.1;
      BLD   103;
      A     I    362.1;
      =     L      0.2;
      BLD   103;
      A     I    362.2;
      =     L      0.3;
      BLD   103;
      A     I    362.3;
      =     L      0.4;
      BLD   103;
      A     I    362.4;
      =     L      0.5;
      BLD   103;
      A     I    362.5;
      =     L      0.6;
      BLD   103;
      A     M   2240.0;
      =     L      2.1;
      BLD   103;
      A     M   2240.1;
      =     L      2.2;
      BLD   103;
      AN    M   2004.0;
      AN    M   2004.1;
      AN    M   6060.1;
      AN    M   6460.0;
      AN    M   6480.0;
      AN    M   2004.2;
      A     M   2000.2;
      =     L      2.3;
      BLD   103;
      A(    ;
      O     I    150.1;
      O     I      0.1;
      )     ;
      =     L      2.5;
      BLD   103;
      A     M      0.5;
      =     L      2.6;
      BLD   103;
      CALL #S704_TL_DC_PIN (
           Enable_Aux               := L      0.0,
           Adv_Amount               := 3,
           Ret_Amount               := 3,
           LS_Adv1                  := L      0.1,
           LS_Ret1                  := L      0.2,
           LS_Adv2                  := L      0.3,
           LS_Ret2                  := L      0.4,
           LS_Adv3                  := L      0.5,
           LS_Ret3                  := L      0.6,
           SOL_Adv                  := L      2.1,
           SOL_Ret                  := L      2.2,
           M_Ready                  := L      2.3,
           T_CHK1                   := T#4S,
           T_CHK2                   := T#4S,
           PB_Error_Rst             := L      2.5,
           M_FLICK                  := L      2.6,
           M_Adv_Err                := M   2250.0,
           M_Ret_Err                := M   2250.1,
           Visu_Adv                 := DB51.DBW  720,
           Visu_Ret                 := DB51.DBW  722);
      NOP   0;
NETWORK
TITLE =
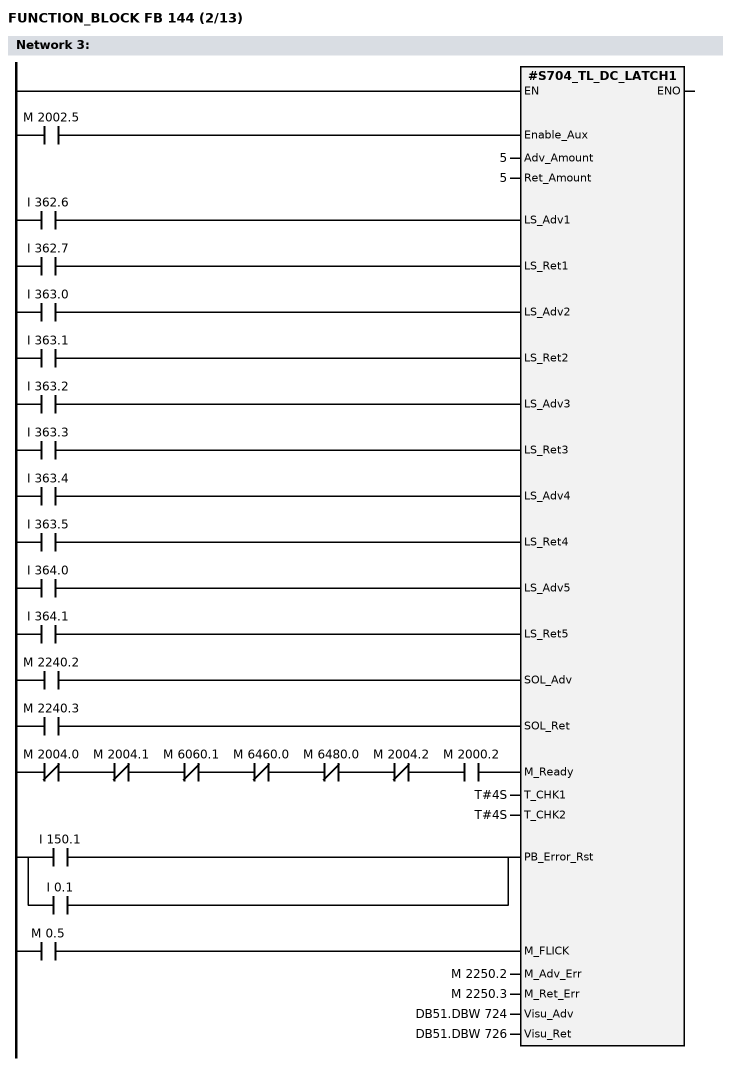

      A     M   2002.5;
      =     L      0.0;
      BLD   103;
      A     I    362.6;
      =     L      0.1;
      BLD   103;
      A     I    362.7;
      =     L      0.2;
      BLD   103;
      A     I    363.0;
      =     L      0.3;
      BLD   103;
      A     I    363.1;
      =     L      0.4;
      BLD   103;
      A     I    363.2;
      =     L      0.5;
      BLD   103;
      A     I    363.3;
      =     L      0.6;
      BLD   103;
      A     I    363.4;
      =     L      0.7;
      BLD   103;
      A     I    363.5;
      =     L      1.0;
      BLD   103;
      A     I    364.0;
      =     L      1.1;
      BLD   103;
      A     I    364.1;
      =     L      1.2;
      BLD   103;
      A     M   2240.2;
      =     L      2.1;
      BLD   103;
      A     M   2240.3;
      =     L      2.2;
      BLD   103;
      AN    M   2004.0;
      AN    M   2004.1;
      AN    M   6060.1;
      AN    M   6460.0;
      AN    M   6480.0;
      AN    M   2004.2;
      A     M   2000.2;
      =     L      2.3;
      BLD   103;
      A(    ;
      O     I    150.1;
      O     I      0.1;
      )     ;
      =     L      2.5;
      BLD   103;
      A     M      0.5;
      =     L      2.6;
      BLD   103;
      CALL #S704_TL_DC_LATCH1 (
           Enable_Aux               := L      0.0,
           Adv_Amount               := 5,
           Ret_Amount               := 5,
           LS_Adv1                  := L      0.1,
           LS_Ret1                  := L      0.2,
           LS_Adv2                  := L      0.3,
           LS_Ret2                  := L      0.4,
           LS_Adv3                  := L      0.5,
           LS_Ret3                  := L      0.6,
           LS_Adv4                  := L      0.7,
           LS_Ret4                  := L      1.0,
           LS_Adv5                  := L      1.1,
           LS_Ret5                  := L      1.2,
           SOL_Adv                  := L      2.1,
           SOL_Ret                  := L      2.2,
           M_Ready                  := L      2.3,
           T_CHK1                   := T#4S,
           T_CHK2                   := T#4S,
           PB_Error_Rst             := L      2.5,
           M_FLICK                  := L      2.6,
           M_Adv_Err                := M   2250.2,
           M_Ret_Err                := M   2250.3,
           Visu_Adv                 := DB51.DBW  724,
           Visu_Ret                 := DB51.DBW  726);
      NOP   0;
NETWORK
TITLE =
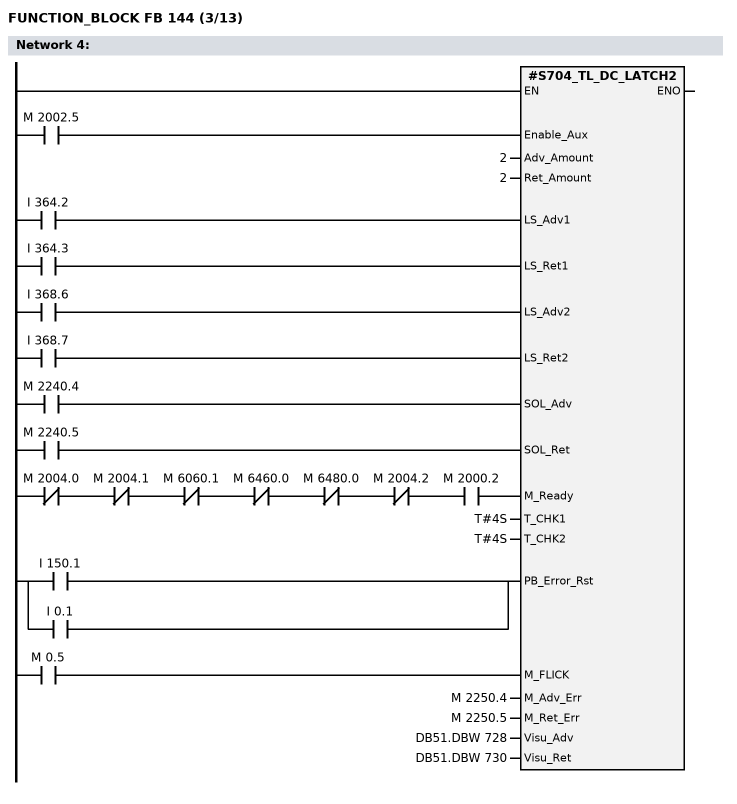

      A     M   2002.5;
      =     L      0.0;
      BLD   103;
      A     I    364.2;
      =     L      0.1;
      BLD   103;
      A     I    364.3;
      =     L      0.2;
      BLD   103;
      A     I    368.6;
      =     L      0.3;
      BLD   103;
      A     I    368.7;
      =     L      0.4;
      BLD   103;
      A     M   2240.4;
      =     L      2.1;
      BLD   103;
      A     M   2240.5;
      =     L      2.2;
      BLD   103;
      AN    M   2004.0;
      AN    M   2004.1;
      AN    M   6060.1;
      AN    M   6460.0;
      AN    M   6480.0;
      AN    M   2004.2;
      A     M   2000.2;
      =     L      2.3;
      BLD   103;
      A(    ;
      O     I    150.1;
      O     I      0.1;
      )     ;
      =     L      2.5;
      BLD   103;
      A     M      0.5;
      =     L      2.6;
      BLD   103;
      CALL #S704_TL_DC_LATCH2 (
           Enable_Aux               := L      0.0,
           Adv_Amount               := 2,
           Ret_Amount               := 2,
           LS_Adv1                  := L      0.1,
           LS_Ret1                  := L      0.2,
           LS_Adv2                  := L      0.3,
           LS_Ret2                  := L      0.4,
           SOL_Adv                  := L      2.1,
           SOL_Ret                  := L      2.2,
           M_Ready                  := L      2.3,
           T_CHK1                   := T#4S,
           T_CHK2                   := T#4S,
           PB_Error_Rst             := L      2.5,
           M_FLICK                  := L      2.6,
           M_Adv_Err                := M   2250.4,
           M_Ret_Err                := M   2250.5,
           Visu_Adv                 := DB51.DBW  728,
           Visu_Ret                 := DB51.DBW  730);
      NOP   0;
NETWORK
TITLE =
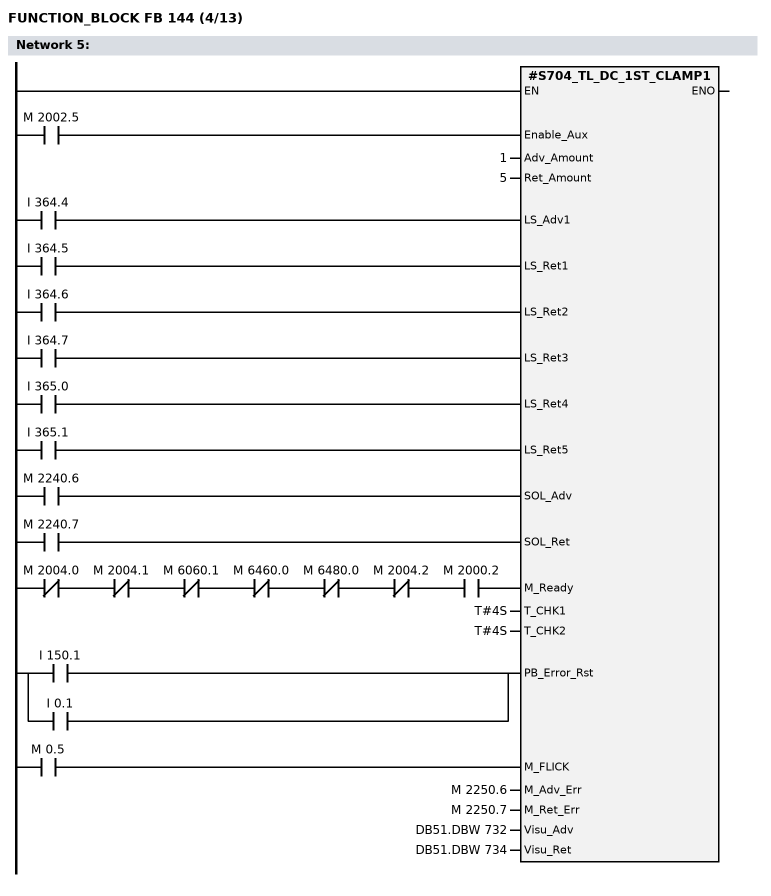

      A     M   2002.5;
      =     L      0.0;
      BLD   103;
      A     I    364.4;
      =     L      0.1;
      BLD   103;
      A     I    364.5;
      =     L      0.2;
      BLD   103;
      A     I    364.6;
      =     L      0.4;
      BLD   103;
      A     I    364.7;
      =     L      0.6;
      BLD   103;
      A     I    365.0;
      =     L      1.0;
      BLD   103;
      A     I    365.1;
      =     L      1.2;
      BLD   103;
      A     M   2240.6;
      =     L      2.1;
      BLD   103;
      A     M   2240.7;
      =     L      2.2;
      BLD   103;
      AN    M   2004.0;
      AN    M   2004.1;
      AN    M   6060.1;
      AN    M   6460.0;
      AN    M   6480.0;
      AN    M   2004.2;
      A     M   2000.2;
      =     L      2.3;
      BLD   103;
      A(    ;
      O     I    150.1;
      O     I      0.1;
      )     ;
      =     L      2.5;
      BLD   103;
      A     M      0.5;
      =     L      2.6;
      BLD   103;
      CALL #S704_TL_DC_1ST_CLAMP1 (
           Enable_Aux               := L      0.0,
           Adv_Amount               := 1,
           Ret_Amount               := 5,
           LS_Adv1                  := L      0.1,
           LS_Ret1                  := L      0.2,
           LS_Ret2                  := L      0.4,
           LS_Ret3                  := L      0.6,
           LS_Ret4                  := L      1.0,
           LS_Ret5                  := L      1.2,
           SOL_Adv                  := L      2.1,
           SOL_Ret                  := L      2.2,
           M_Ready                  := L      2.3,
           T_CHK1                   := T#4S,
           T_CHK2                   := T#4S,
           PB_Error_Rst             := L      2.5,
           M_FLICK                  := L      2.6,
           M_Adv_Err                := M   2250.6,
           M_Ret_Err                := M   2250.7,
           Visu_Adv                 := DB51.DBW  732,
           Visu_Ret                 := DB51.DBW  734);
      NOP   0;
NETWORK
TITLE =
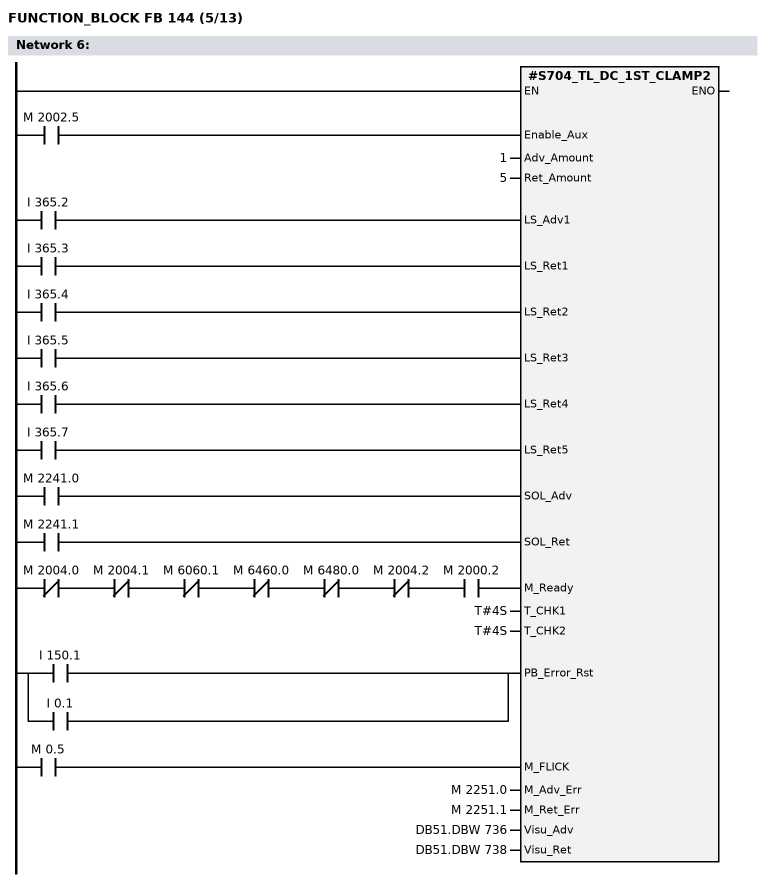

      A     M   2002.5;
      =     L      0.0;
      BLD   103;
      A     I    365.2;
      =     L      0.1;
      BLD   103;
      A     I    365.3;
      =     L      0.2;
      BLD   103;
      A     I    365.4;
      =     L      0.4;
      BLD   103;
      A     I    365.5;
      =     L      0.6;
      BLD   103;
      A     I    365.6;
      =     L      1.0;
      BLD   103;
      A     I    365.7;
      =     L      1.2;
      BLD   103;
      A     M   2241.0;
      =     L      2.1;
      BLD   103;
      A     M   2241.1;
      =     L      2.2;
      BLD   103;
      AN    M   2004.0;
      AN    M   2004.1;
      AN    M   6060.1;
      AN    M   6460.0;
      AN    M   6480.0;
      AN    M   2004.2;
      A     M   2000.2;
      =     L      2.3;
      BLD   103;
      A(    ;
      O     I    150.1;
      O     I      0.1;
      )     ;
      =     L      2.5;
      BLD   103;
      A     M      0.5;
      =     L      2.6;
      BLD   103;
      CALL #S704_TL_DC_1ST_CLAMP2 (
           Enable_Aux               := L      0.0,
           Adv_Amount               := 1,
           Ret_Amount               := 5,
           LS_Adv1                  := L      0.1,
           LS_Ret1                  := L      0.2,
           LS_Ret2                  := L      0.4,
           LS_Ret3                  := L      0.6,
           LS_Ret4                  := L      1.0,
           LS_Ret5                  := L      1.2,
           SOL_Adv                  := L      2.1,
           SOL_Ret                  := L      2.2,
           M_Ready                  := L      2.3,
           T_CHK1                   := T#4S,
           T_CHK2                   := T#4S,
           PB_Error_Rst             := L      2.5,
           M_FLICK                  := L      2.6,
           M_Adv_Err                := M   2251.0,
           M_Ret_Err                := M   2251.1,
           Visu_Adv                 := DB51.DBW  736,
           Visu_Ret                 := DB51.DBW  738);
      NOP   0;
NETWORK
TITLE =
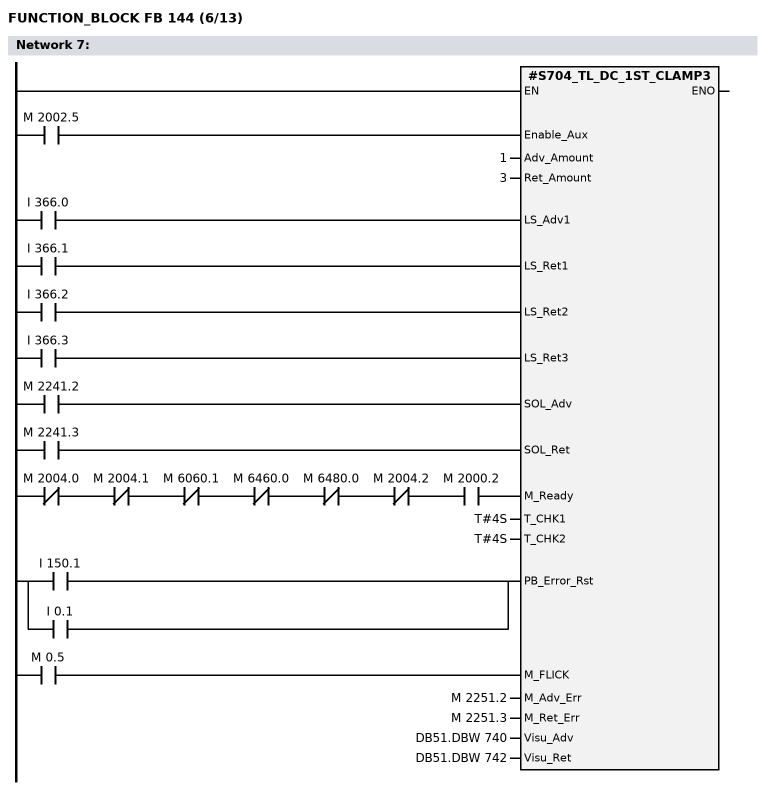

      A     M   2002.5;
      =     L      0.0;
      BLD   103;
      A     I    366.0;
      =     L      0.1;
      BLD   103;
      A     I    366.1;
      =     L      0.2;
      BLD   103;
      A     I    366.2;
      =     L      0.4;
      BLD   103;
      A     I    366.3;
      =     L      0.6;
      BLD   103;
      A     M   2241.2;
      =     L      2.1;
      BLD   103;
      A     M   2241.3;
      =     L      2.2;
      BLD   103;
      AN    M   2004.0;
      AN    M   2004.1;
      AN    M   6060.1;
      AN    M   6460.0;
      AN    M   6480.0;
      AN    M   2004.2;
      A     M   2000.2;
      =     L      2.3;
      BLD   103;
      A(    ;
      O     I    150.1;
      O     I      0.1;
      )     ;
      =     L      2.5;
      BLD   103;
      A     M      0.5;
      =     L      2.6;
      BLD   103;
      CALL #S704_TL_DC_1ST_CLAMP3 (
           Enable_Aux               := L      0.0,
           Adv_Amount               := 1,
           Ret_Amount               := 3,
           LS_Adv1                  := L      0.1,
           LS_Ret1                  := L      0.2,
           LS_Ret2                  := L      0.4,
           LS_Ret3                  := L      0.6,
           SOL_Adv                  := L      2.1,
           SOL_Ret                  := L      2.2,
           M_Ready                  := L      2.3,
           T_CHK1                   := T#4S,
           T_CHK2                   := T#4S,
           PB_Error_Rst             := L      2.5,
           M_FLICK                  := L      2.6,
           M_Adv_Err                := M   2251.2,
           M_Ret_Err                := M   2251.3,
           Visu_Adv                 := DB51.DBW  740,
           Visu_Ret                 := DB51.DBW  742);
      NOP   0;
NETWORK
TITLE =
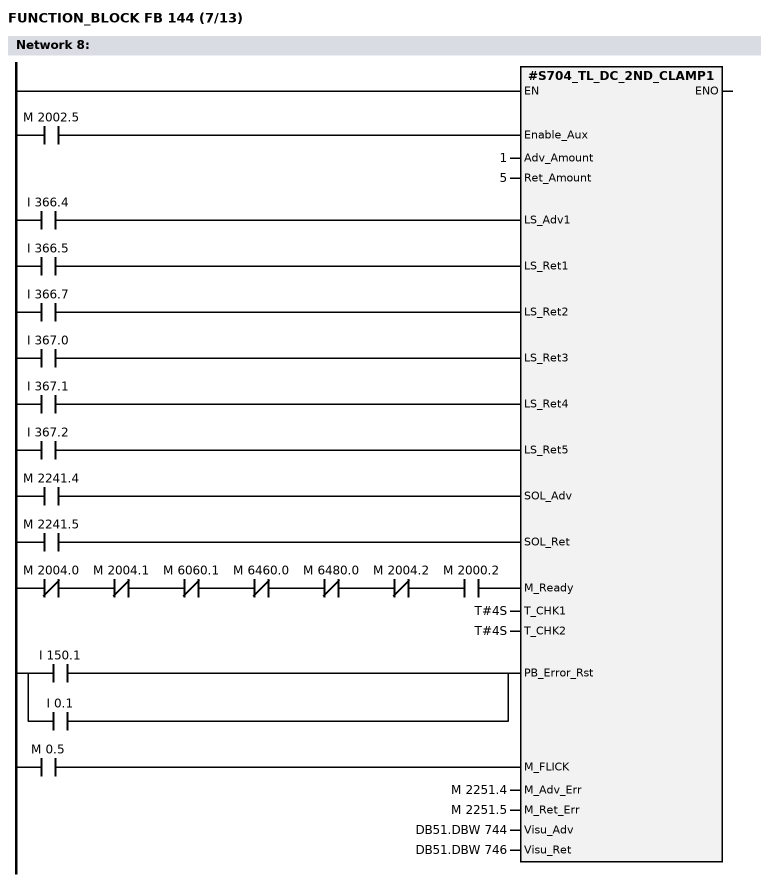

      A     M   2002.5;
      =     L      0.0;
      BLD   103;
      A     I    366.4;
      =     L      0.1;
      BLD   103;
      A     I    366.5;
      =     L      0.2;
      BLD   103;
      A     I    366.7;
      =     L      0.4;
      BLD   103;
      A     I    367.0;
      =     L      0.6;
      BLD   103;
      A     I    367.1;
      =     L      1.0;
      BLD   103;
      A     I    367.2;
      =     L      1.2;
      BLD   103;
      A     M   2241.4;
      =     L      2.1;
      BLD   103;
      A     M   2241.5;
      =     L      2.2;
      BLD   103;
      AN    M   2004.0;
      AN    M   2004.1;
      AN    M   6060.1;
      AN    M   6460.0;
      AN    M   6480.0;
      AN    M   2004.2;
      A     M   2000.2;
      =     L      2.3;
      BLD   103;
      A(    ;
      O     I    150.1;
      O     I      0.1;
      )     ;
      =     L      2.5;
      BLD   103;
      A     M      0.5;
      =     L      2.6;
      BLD   103;
      CALL #S704_TL_DC_2ND_CLAMP1 (
           Enable_Aux               := L      0.0,
           Adv_Amount               := 1,
           Ret_Amount               := 5,
           LS_Adv1                  := L      0.1,
           LS_Ret1                  := L      0.2,
           LS_Ret2                  := L      0.4,
           LS_Ret3                  := L      0.6,
           LS_Ret4                  := L      1.0,
           LS_Ret5                  := L      1.2,
           SOL_Adv                  := L      2.1,
           SOL_Ret                  := L      2.2,
           M_Ready                  := L      2.3,
           T_CHK1                   := T#4S,
           T_CHK2                   := T#4S,
           PB_Error_Rst             := L      2.5,
           M_FLICK                  := L      2.6,
           M_Adv_Err                := M   2251.4,
           M_Ret_Err                := M   2251.5,
           Visu_Adv                 := DB51.DBW  744,
           Visu_Ret                 := DB51.DBW  746);
      NOP   0;
NETWORK
TITLE =
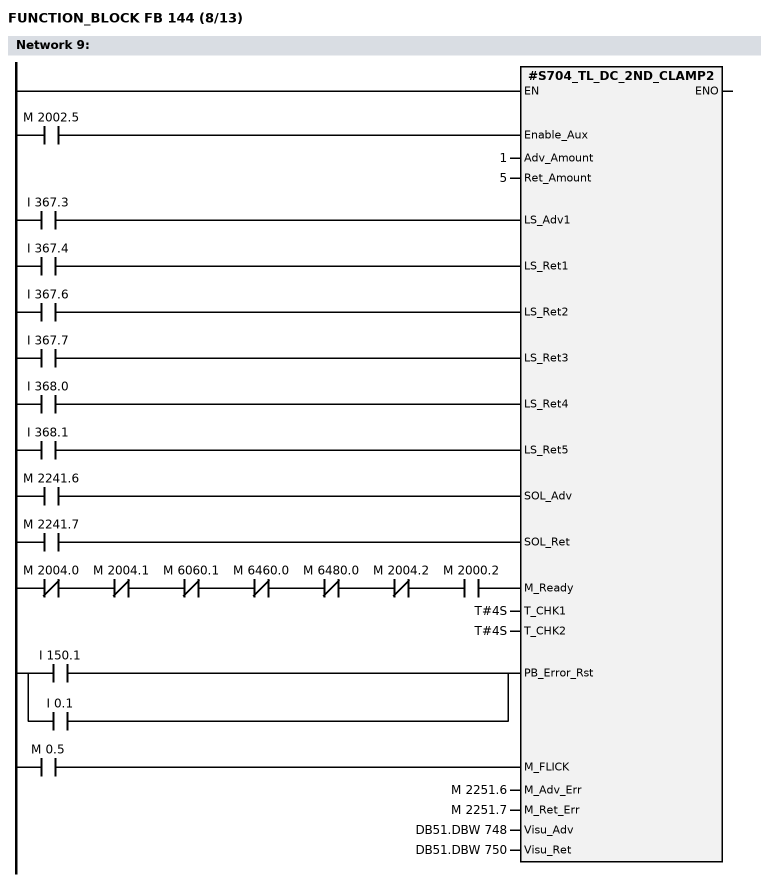

